	bEnableLuxEvent				: BOOL;
	eEventPriorityBrightness	: E_DALIEventPriority := E_DALIEVENTPRIORITY.Middle;
	nDeadtimeTimerBrightness	: WORD := 1500; // Value in ms, Predefined Value of DALI Standard
	nHysteresisBrightness		: BYTE := 2; // Value in %
	nHysteresisMinBrightness	: BYTE := 10; // Absolute Value, depending on the manufacturer specific resolution
	nReportTimerBrightness		: BYTE := 120; // Value in s, Preset manufacturer value
*)

	//stDaliSetup: SH_Light.ST_DALI_RoomSetup;

END_VAR

VAR CONSTANT
	Sensor_DALI_LINE_NUM: BYTE := 3;
	arrDALI_LINE_NUM_LIGHT: ARRAY[1..2] OF BYTE := [2,1]; //korrekt rækkefølge nødvendig
	arrDALI_LINE_NUM_PENDANTS: ARRAY[1..2] OF BYTE := [0,0]; //korrekt rækkefølge nødvendig. 0 = ingen pendler
END_VAR
VAR PERSISTENT
	stPirSensorData: SH_Light.ST_DALI_Sensor;
	arrstTuneDataGruppe: ARRAY [1..2] OF SH_Light.ST_TuneData_EX;
END_VAR

A_Buttons();
A_LightCtrl();
A_Sensor();

ACTION A_Buttons:
bTopButtonZone1		:= GVL_EnOcean.strEnOceanSwitch_Gang_4_330.bT2_OFF OR bTopButtonZone1_Visu;
bBottomButtonZone1	:= GVL_EnOcean.strEnOceanSwitch_Gang_4_330.bT2_ON OR bBottomButtonZone1_Visu;
END_ACTION

ACTION A_LightCtrl:
bNeighborRoomsPir	:= P_Gang_4_308.stPirSensorData.bPrc      OR
						P_Rum_4_324.stPirSensorData.bPrc      OR
						P_Rum_4_325.stPirSensorData.bPrc      OR
						P_Rum_4_329.stPirSensorData.bPrc;


//gruppe 3
arrfbLysGruppe[1]( 
	nZoneID:= 1, 
	bButtonZone1:= bTopButtonZone1,
	bBottomButtonZone1 := bBottomButtonZone1, 
	bButtonZone2:= bButtonZone2,
	bNeighborRoomsPir	:=	bNeighborRoomsPir,
	fLuxOn:= fLuxOn, 
	fLuxDim:= fLuxDim, 
	tPIRDim:= tPIRDim, 
	tPIROff:= tPIROff, 
	fOffsetSec:= fOffsetSec, 
	bReInit:= , 
	stDaliSetup:= arrstDaliSetupGruppe[1], 
	ipCommunication_Prim:= P_DALI_Background.arrfbKL6821Communication[arrDALI_LINE_NUM_LIGHT[1]], 
	ipCommunication_Sec:= P_DALI_Background.arrfbKL6821Communication[arrDALI_LINE_NUM_LIGHT[1]], //samme som lyslinjen, hvis den ikke eksisterer
	ipCommunication_Supl:= P_DALI_Background.arrfbKL6821Communication[arrDALI_LINE_NUM_LIGHT[1]],//samme som lyslinjen, hvis den ikke eksisterer 
	fMinOutputPowerLevelRoom:= 15, 
	fMaxOutputPowerLevelRoom:= 100, 
	nCycleTimeInMS:= 10 , 
	bRunTuning:= arrRunTuningGruppe[1], 
	bOccupiedRoom=> , 
	bError_Prim=> , 
	nError_Prim=> , 
	stTuneData:=arrstTuneDataGruppe[1] , 
	stPirSensorData:= stPirSensorData, 					//samme sensordata
	stLiveData:= arrstLiveDataGruppe[1]);

//gruppe 13
arrfbLysGruppe[2]( 
	nZoneID:= 1, 
	bButtonZone1:= bTopButtonZone1,
	bBottomButtonZone1 := bBottomButtonZone1, 
	bButtonZone2:= bButtonZone2,
	bNeighborRoomsPir	:=	bNeighborRoomsPir,
	fLuxOn:= fLuxOn, 
	fLuxDim:= fLuxDim, 
	tPIRDim:= tPIRDim, 
	tPIROff:= tPIROff, 
	fOffsetSec:= fOffsetSec, 
	bReInit:= , 
	stDaliSetup:= arrstDaliSetupGruppe[2], 
	ipCommunication_Prim:= P_DALI_Background.arrfbKL6821Communication[arrDALI_LINE_NUM_LIGHT[2]], 
	ipCommunication_Sec:= P_DALI_Background.arrfbKL6821Communication[arrDALI_LINE_NUM_LIGHT[2]], //samme som lyslinjen, hvis den ikke eksisterer
	ipCommunication_Supl:= P_DALI_Background.arrfbKL6821Communication[arrDALI_LINE_NUM_LIGHT[2]], //samme som lyslinjen, hvis den ikke eksisterer 
	fMinOutputPowerLevelRoom:= 15, 
	fMaxOutputPowerLevelRoom:= 100, 
	nCycleTimeInMS:= 10 , 
	bRunTuning:= arrRunTuningGruppe[2], 
	bOccupiedRoom=> , 
	bError_Prim=> , 
	nError_Prim=> , 
	stTuneData:=arrstTuneDataGruppe[2] , 
	stPirSensorData:= stPirSensorData, 					//samme sensordata
	stLiveData:= arrstLiveDataGruppe[2]);
END_ACTION

ACTION A_Sensor:

fbSensor.ipCommunication := P_DALI_Background.arrfbKL6821Communication[Sensor_DALI_LINE_NUM];

//only 1 sensor
fbSensor(
	byShrtAdr:= bySensorAddr,
	bInitialize:= bInitialize, 
	DALI_LINE_NUM:= Sensor_DALI_LINE_NUM, 
 	//bCancelHoldTimerOccupancy:= bCancelHoldTimerOccupancy, 
	stSensorSetup := stDaliSensorSetup,
	bInitErr=> bInitErr, 
	bInitDone=> bInitDone,
	stPirSensorData:= stPirSensorData, 
	arrSensorScales:= arrSensorScales);


(*//several sensors	
fbSensor(
	arrShrtAdr:= arrSensorAddr,
	bInitialize:= bInitialize, 
	DALI_LINE_NUM:= Sensor_DALI_LINE_NUM, 
 	//bCancelHoldTimerOccupancy:= bCancelHoldTimerOccupancy, 
	stSensorSetup := stDaliSensorSetup,
	arrInitErr=> arrInitErr, 
	arrInitDone=> arrInitDone,
	stPirSensorData:= stPirSensorData, 
	arrSensorScales:= arrSensorScales);
	*)
END_ACTION

END_PROGRAM

// ---- POUs/Alle_Rum/Gange/Gang_4_308_2linjerLampe/P_Gang_4_308.TcPOU
PROGRAM P_Gang_4_308
VAR
(*Gangen består af to lysgrupper - 5 og 14 - på to forskellige DALI-linjer - 2 og 1 henh..
Begge grupper afhænger af samme PIR-input - pir-adr. 6, 7, 8, 9 og 10 - på DALI-linje 2.
Derfor oprettes to adskilte reguleringer med samme PV. Dvs., at knapfunktion og pirfunktion forbliver den samme.

En anden del af af hele gangen styres fra AH4_3. De to dele nabostyres med PIR-signaler over modbus-kommunikation*)

	arrfbLysGruppe			: ARRAY [1..2] OF FB_Light_Type_B;
	arrstDaliSetupGruppe	: ARRAY[1..2] OF SH_Light.ST_DALI_RoomSetup := 
	
													[(	byShrtAdr_Prim := 29, 
														byGrpAdr_Prim := 5, 
														eMod_Prim := E_DALIAddressType.Group, 
														byShrtAdr_Sec := 1, 
														byGrpAdr_Sec := 1, 
														eMod_Sec := E_DALIAddressType.Short, 
														byShrtAdr_Supl := 1, 
														DALI_LINE_NUM_PRIM := arrDALI_LINE_NUM_LIGHT[1], 
														DALI_LINE_NUM_SEC := 0, //0 = ingen zonestyring/vinduerække
														DALI_LINE_NUM_SUPL := arrDALI_LINE_NUM_PENDANTS[1]),
														
													(	byShrtAdr_Prim := 51, 
														byGrpAdr_Prim := 14, 
														eMod_Prim := E_DALIAddressType.Group, 
														byShrtAdr_Sec := 1, 
														byGrpAdr_Sec := 1, 
														eMod_Sec := E_DALIAddressType.Short, 
														byShrtAdr_Supl := 1, 
														DALI_LINE_NUM_PRIM := arrDALI_LINE_NUM_LIGHT[2], 
														DALI_LINE_NUM_SEC := 0, 
														DALI_LINE_NUM_SUPL := arrDALI_LINE_NUM_PENDANTS[2])];
														
	arrstLiveDataGruppe		: ARRAY [1..2] OF SH_Light.ST_LiveData;
	//stLiveData AT %MB22	: SH_Light.ST_LiveData;
	
	arrRunTuningGruppe: ARRAY[1..2] OF BOOL;
	
	
	
	bTopButtonZone1			: BOOL;
	bTopButtonZone1_Visu	: BOOL;
	bBottomButtonZone1		: BOOL;
	bBottomButtonZone1_Visu	: BOOL;
	bButtonZone2			: BOOL;
	bNeighborRoomsPir		: BOOL;
	fLuxOn					: REAL := 500;
	fLuxDim					: REAL := 200;
	tPIRDim					: TIME := T#15M;
	tPIROff					: TIME := T#30M;
	fOffsetSec				: REAL := 20;



// Sensor Settings
	//fbSensor					: SH_Light.FB_NIKO_P46xx_1Pcs;
	fbSensor					: SH_Light.FB_NIKO_P46xx_3Pcs;
	//bySensorAddr				: BYTE := 17;
	arrSensorAddr				: ARRAY[1..3] OF BYTE := [7,8,9];
	bInitialize					: BOOL := TRUE;
	stDaliSensorSetup			: ST_DALI_NIKOP46SetupData;
	//bInitErr					: BOOL;
	//bInitDone					: BOOL;
	arrInitErr					: ARRAY [1..3] OF BOOL;
	arrInitDone					: ARRAY [1..3] OF BOOL;
	arrSensorScales				: ARRAY [1..10] OF SH_Light.ST_DALI_SensorScaleMode := [	(fMeassureMaxSensor := 1023, fReadMaxSensor := 1023),
																							(fMeassureMaxSensor := 1023, fReadMaxSensor := 1023),
																							(fMeassureMaxSensor := 1023, fReadMaxSensor := 1023),																						
																						7(())];
	bCancelHoldTimerOccupancy	: BOOL;
(*	eEventPriorityOccupancy		: E_DALIEventPriority := E_DALIEVENTPRIORITY.Middle;
	nHoldTimerOccupancy			: WORD := 5; // Value in s. 	
	nReportTimerOccupancy		: BYTE := 120; // Value in s, Preset manufacturer value
	nDeadtimeTimerOccupancy		: WORD := 100; // Value in ms, Predefined Value of DALI Standard
	bCancelHoldTimerOccupancy	: BOOL;
	nSensitivityOccupancy		: BYTE:= 3; //setting Sensivity (0..4) 0 (Off), 1 (Min), 2(Low), 3(High) and 4 (Max)

	bEnableLuxEvent				: BOOL;
	eEventPriorityBrightness	: E_DALIEventPriority := E_DALIEVENTPRIORITY.Middle;
	nDeadtimeTimerBrightness	: WORD := 1500; // Value in ms, Predefined Value of DALI Standard
	nHysteresisBrightness		: BYTE := 2; // Value in %
	nHysteresisMinBrightness	: BYTE := 10; // Absolute Value, depending on the manufacturer specific resolution
	nReportTimerBrightness		: BYTE := 120; // Value in s, Preset manufacturer value
*)


END_VAR

VAR CONSTANT
	Sensor_DALI_LINE_NUM: BYTE := 3;
	arrDALI_LINE_NUM_LIGHT: ARRAY[1..2] OF BYTE := [2,1]; //korrekt rækkefølge nødvendig
	arrDALI_LINE_NUM_PENDANTS: ARRAY[1..2] OF BYTE := [0,0]; //korrekt rækkefølge nødvendig. 0 = ingen pendler
END_VAR
VAR PERSISTENT
	stPirSensorData: SH_Light.ST_DALI_Sensor;
	arrstTuneDataGruppe: ARRAY [1..2] OF SH_Light.ST_TuneData_EX;
END_VAR

A_Buttons();
A_LightCtrl();
A_Sensor();

ACTION A_Buttons:
bTopButtonZone1		:= bTopButtonZone1_Visu;
bBottomButtonZone1	:= bBottomButtonZone1_Visu;
END_ACTION

ACTION A_LightCtrl:
bNeighborRoomsPir	:=  
						P_Rum_4_324.stPirSensorData.bPrc OR
				     	P_Gang_4_330.stPirSensorData.bPrc OR
						P_Gang_4_334A.stPirSensorData.bPrc OR
                        P_Gang_5_338.stPirSensorData.bPrc;

//gruppe 5
arrfbLysGruppe[1]( 
	nZoneID:= 1, 
	bButtonZone1:= bTopButtonZone1,
	bBottomButtonZone1 := bBottomButtonZone1, 
	bButtonZone2:= bButtonZone2,
	bNeighborRoomsPir	:=	bNeighborRoomsPir,
	fLuxOn:= fLuxOn, 
	fLuxDim:= fLuxDim, 
	tPIRDim:= tPIRDim, 
	tPIROff:= tPIROff, 
	fOffsetSec:= fOffsetSec, 
	bReInit:= , 
	stDaliSetup:= arrstDaliSetupGruppe[1], 
	ipCommunication_Prim:= P_DALI_Background.arrfbKL6821Communication[arrDALI_LINE_NUM_LIGHT[1]], 
	ipCommunication_Sec:= P_DALI_Background.arrfbKL6821Communication[arrDALI_LINE_NUM_LIGHT[1]], //samme som lyslinjen, hvis den ikke eksisterer
	ipCommunication_Supl:= P_DALI_Background.arrfbKL6821Communication[arrDALI_LINE_NUM_LIGHT[1]],//samme som lyslinjen, hvis den ikke eksisterer 
	fMinOutputPowerLevelRoom:= 15, 
	fMaxOutputPowerLevelRoom:= 100, 
	nCycleTimeInMS:= 10 , 
	bRunTuning:= arrRunTuningGruppe[1], 
	bOccupiedRoom=> , 
	bError_Prim=> , 
	nError_Prim=> , 
	stTuneData:=arrstTuneDataGruppe[1] , 
	stPirSensorData:= stPirSensorData, 					//samme sensordata
	stLiveData:= arrstLiveDataGruppe[1]);

//gruppe 14	
arrfbLysGruppe[2]( 
	nZoneID:= 1, 
	bButtonZone1:= bTopButtonZone1,
	bBottomButtonZone1 := bBottomButtonZone1, 
	bButtonZone2:= bButtonZone2,
	bNeighborRoomsPir	:=	bNeighborRoomsPir,
	fLuxOn:= fLuxOn, 
	fLuxDim:= fLuxDim, 
	tPIRDim:= tPIRDim, 
	tPIROff:= tPIROff, 
	fOffsetSec:= fOffsetSec, 
	bReInit:= , 
	stDaliSetup:= arrstDaliSetupGruppe[2], 
	ipCommunication_Prim:= P_DALI_Background.arrfbKL6821Communication[arrDALI_LINE_NUM_LIGHT[2]], 
	ipCommunication_Sec:= P_DALI_Background.arrfbKL6821Communication[arrDALI_LINE_NUM_LIGHT[2]], //samme som lyslinjen, hvis den ikke eksisterer
	ipCommunication_Supl:= P_DALI_Background.arrfbKL6821Communication[arrDALI_LINE_NUM_LIGHT[2]], //samme som lyslinjen, hvis den ikke eksisterer 
	fMinOutputPowerLevelRoom:= 15, 
	fMaxOutputPowerLevelRoom:= 100, 
	nCycleTimeInMS:= 10 , 
	bRunTuning:= arrRunTuningGruppe[2], 
	bOccupiedRoom=> , 
	bError_Prim=> , 
	nError_Prim=> , 
	stTuneData:=arrstTuneDataGruppe[2] , 
	stPirSensorData:= stPirSensorData, 					//samme sensordata
	stLiveData:= arrstLiveDataGruppe[2]);
END_ACTION

ACTION A_Sensor:

fbSensor.ipCommunication := P_DALI_Background.arrfbKL6821Communication[Sensor_DALI_LINE_NUM];

(*//only 1 sensor
fbSensor(
	byShrtAdr:= bySensorAddr,
	bInitialize:= bInitialize, 
	DALI_LINE_NUM:= Sensor_DALI_LINE_NUM, 
 	//bCancelHoldTimerOccupancy:= bCancelHoldTimerOccupancy, 
	stSensorSetup := stDaliSensorSetup,
	bInitErr=> bInitErr, 
	bInitDone=> bInitDone,
	stPirSensorData:= stPirSensorData, 
	arrSensorScales:= arrSensorScales);
	*)

//several sensors	
fbSensor(
	arrShrtAdr:= arrSensorAddr,
	bInitialize:= bInitialize, 
	DALI_LINE_NUM:= Sensor_DALI_LINE_NUM, 
 	//bCancelHoldTimerOccupancy:= bCancelHoldTimerOccupancy, 
	stSensorSetup := stDaliSensorSetup,
	arrInitErr=> arrInitErr, 
	arrInitDone=> arrInitDone,
	stPirSensorData:= stPirSensorData, 
	arrSensorScales:= arrSensorScales);
END_ACTION

END_PROGRAM

// ---- POUs/Alle_Rum/Gange/Gang_4_310A/P_Gang_4_310A.TcPOU
PROGRAM P_Gang_4_310A
VAR
//Light

(*Toiletgangen er oprettet som type B i tilfælde af, at gangen skal nabostyres af toiletter mv. i fremtiden.
For nu er der ingen pirsignaler fra toiletter til PLC*)

	fbLys		: FB_Light_Type_B;
	
	stDaliSetup	: SH_Light.ST_DALI_RoomSetup := (		byShrtAdr_Prim := 34, 
														byGrpAdr_Prim := 5, 
														eMod_Prim := E_DALIAddressType.Group, 
														byShrtAdr_Sec := 1, 
														byGrpAdr_Sec := 1, 
														eMod_Sec := E_DALIAddressType.Short, 
														byShrtAdr_Supl := 1, 
														DALI_LINE_NUM_PRIM := DALI_LINE_NUM_LIGHT, 
														DALI_LINE_NUM_SEC := 0, 
														DALI_LINE_NUM_SUPL := DALI_LINE_NUM_PENDANTS);
	stLiveData				: SH_Light.ST_LiveData;
	//stLiveData AT %MB22	: SH_Light.ST_LiveData;
	bTopButtonZone1			: BOOL;
	bTopButtonZone1_Visu		: BOOL;
	bBottomButtonZone1		: BOOL;
	bBottomButtonZone1_Visu	: BOOL;
	bButtonZone2			: BOOL;
	bNeighborRoomsPir		: BOOL;
	fLuxOn					: REAL := 500;
	fLuxDim					: REAL := 200;
	tPIRDim					: TIME := T#15M;
	tPIROff					: TIME := T#30M;
	fOffsetSec				: REAL := 20;

	bRunTuning: BOOL;

// Sensor Settings
	fbSensor					: SH_Light.FB_NIKO_P46xx_1Pcs;	
	//fbSensor					: SH_Light.FB_NIKO_P46xx_2Pcs;
	bySensorAddr				: BYTE := 1;
	//arrSensorAddr				: ARRAY[1..2] OF BYTE := [12,13];
	bInitialize					: BOOL := TRUE;
	stDaliSensorSetup			: ST_DALI_NIKOP46SetupData;
	bInitErr					: BOOL;
	bInitDone					: BOOL;
	//arrInitErr					: ARRAY [1..2] OF BOOL;
	//arrInitDone					: ARRAY [1..2] OF BOOL;
	arrSensorScales				: ARRAY [1..10] OF SH_Light.ST_DALI_SensorScaleMode := [	(fMeassureMaxSensor := 1023, fReadMaxSensor := 1023),
																						9(())];
	bCancelHoldTimerOccupancy	: BOOL;
(*	eEventPriorityOccupancy		: E_DALIEventPriority := E_DALIEVENTPRIORITY.Middle;
	nHoldTimerOccupancy			: WORD := 5; // Value in s. 	
	nReportTimerOccupancy		: BYTE := 120; // Value in s, Preset manufacturer value
	nDeadtimeTimerOccupancy		: WORD := 100; // Value in ms, Predefined Value of DALI Standard
	bCancelHoldTimerOccupancy	: BOOL;
	nSensitivityOccupancy		: BYTE:= 3; //setting Sensivity (0..4) 0 (Off), 1 (Min), 2(Low), 3(High) and 4 (Max)

	bEnableLuxEvent				: BOOL;
	eEventPriorityBrightness	: E_DALIEventPriority := E_DALIEVENTPRIORITY.Middle;
	nDeadtimeTimerBrightness	: WORD := 1500; // Value in ms, Predefined Value of DALI Standard
	nHysteresisBrightness		: BYTE := 2; // Value in %
	nHysteresisMinBrightness	: BYTE := 10; // Absolute Value, depending on the manufacturer specific resolution
	nReportTimerBrightness		: BYTE := 120; // Value in s, Preset manufacturer value
*)

END_VAR

VAR CONSTANT
	Sensor_DALI_LINE_NUM	: BYTE := 3;
	DALI_LINE_NUM_LIGHT		: BYTE := 3;
	DALI_LINE_NUM_PENDANTS	: BYTE := 0;
END_VAR
VAR PERSISTENT
	stPirSensorData: SH_Light.ST_DALI_Sensor;
	stTuneData: SH_Light.ST_TuneData_EX;
END_VAR

A_Buttons();
A_LightCtrl();
A_Sensor();

ACTION A_Buttons:
bTopButtonZone1		:=  bTopButtonZone1_Visu;
bBottomButtonZone1	:=  bBottomButtonZone1_Visu;
END_ACTION

ACTION A_LightCtrl:
bNeighborRoomsPir	:= 0; //evt. nabostyring
						
fbLys(
	nZoneID:= 1, 
	bButtonZone1:= bTopButtonZone1,
	bBottomButtonZone1 := bBottomButtonZone1, 
	bButtonZone2:= bButtonZone2,
	bNeighborRoomsPir	:=	bNeighborRoomsPir,
	fLuxOn:= fLuxOn, 
	fLuxDim:= fLuxDim, 
	tPIRDim:= tPIRDim, 
	tPIROff:= tPIROff, 
	fOffsetSec:= fOffsetSec, 
	bReInit:= , 
	stDaliSetup:= stDaliSetup, 
	ipCommunication_Prim:= P_DALI_Background.arrfbKL6821Communication[DALI_LINE_NUM_LIGHT], 
	ipCommunication_Sec:= P_DALI_Background.arrfbKL6821Communication[DALI_LINE_NUM_LIGHT], 
	ipCommunication_Supl:= P_DALI_Background.arrfbKL6821Communication[DALI_LINE_NUM_LIGHT], 
	fMinOutputPowerLevelRoom:= 15, 
	fMaxOutputPowerLevelRoom:= 100, 
	nCycleTimeInMS:= 10 , 
	bRunTuning:= bRunTuning, 
	bOccupiedRoom=> , 
	bError_Prim=> , 
	nError_Prim=> , 
	stTuneData:=stTuneData , 
	stPirSensorData:= stPirSensorData, 
	stLiveData:= stLiveData);
END_ACTION

ACTION A_Sensor:

fbSensor.ipCommunication := P_DALI_Background.arrfbKL6821Communication[Sensor_DALI_LINE_NUM];

//Only 1 sensor
fbSensor(
	byShrtAdr:= bySensorAddr,
	bInitialize:= bInitialize, 
	DALI_LINE_NUM:= Sensor_DALI_LINE_NUM, 
 	//bCancelHoldTimerOccupancy:= bCancelHoldTimerOccupancy, 
	stSensorSetup := stDaliSensorSetup,
	bInitErr=> bInitErr, 
	bInitDone=> bInitDone,
	stPirSensorData:= stPirSensorData, 
	arrSensorScales:= arrSensorScales);

(*//Several sensors
fbSensor(
	arrShrtAdr:= arrSensorAddr,
	bInitialize:= bInitialize, 
	DALI_LINE_NUM:= Sensor_DALI_LINE_NUM, 
 	//bCancelHoldTimerOccupancy:= bCancelHoldTimerOccupancy, 
	stSensorSetup := stDaliSensorSetup,
	arrInitErr=> arrInitErr, 
	arrInitDone=> arrInitDone,
	stPirSensorData:= stPirSensorData, 
	arrSensorScales:= arrSensorScales);
	*)
END_ACTION

END_PROGRAM

// ---- POUs/Alle_Rum/Rum_Med_DALI_Pir/P_Lys_Grp0.TcPOU
PROGRAM P_Lys_Grp0
VAR
	fbLight_GRP0: FB_DALILgtActr_EX;
	eMod: SH_Light.E_DALIAddressType := SH_Light.E_DALIAddressType.Group;
	fSttupCtrlVal: REAL;
	fMinCtrlVal: REAL := 0;
	fMaxCtrlVal: REAL := 100;
	fLgtOffset: REAL := 5;
	eFadeTime: SH_Light.E_DALIFadeTime := SH_Light.E_DALIFadeTime.T02000ms;
	eFadeRate: SH_Light.E_DALIFadeRate := SH_Light.E_DALIFadeRate.N063StepsPerSec;
	uiBlinkTi: UINT := 2;
	uiOffDly: UINT := 0;
	uiPollActLgtLvl: UINT := 30;
	bReInit: BOOL;
	nCycleTimeInMS: UDINT := 10;
	stLgtCmd: SH_Light.ST_LgtCmd;
END_VAR

VAR CONSTANT
	DALI_LINE_NUM: BYTE := 1;
END_VAR

fbLight_GRP0.ipDALICommunication := P_DALI_Background.arrfbKL6821Communication[DALI_LINE_NUM];
fbLight_GRP0(
    byShrtAdr := 6,
    byGrpAdr := 1,
    eMod := eMod,
    fSttupCtrlVal := fSttupCtrlVal,
    fMinCtrlVal := fMinCtrlVal,
    fMaxCtrlVal := fMaxCtrlVal,
    fLgtOffset := fLgtOffset,
    eFadeTime := eFadeTime,
    eFadeRate := eFadeRate,
    uiBlinkTi := uiBlinkTi,
    uiOffDly := uiOffDly,
    uiPollActLgtLvl := uiPollActLgtLvl,
    bReInit := bReInit,
    nCycleTimeInMS := nCycleTimeInMS,
    stLgtCmd := stLgtCmd,
    DALI_LINE_NUM := DALI_LINE_NUM); // FB_DALILgtActr_EX

END_PROGRAM

// ---- POUs/Alle_Rum/Rum_Med_DALI_Pir/Rum_5_341/P_Rum_5_341.TcPOU
PROGRAM P_Rum_5_341
VAR
//Light

	fbLys		: FB_Light_Type_A;
	
	stDaliSetup	: SH_Light.ST_DALI_RoomSetup := (		byShrtAdr_Prim := 5, 
														byGrpAdr_Prim := 2, 
														eMod_Prim := E_DALIAddressType.Group, 
														byShrtAdr_Sec := 1, 
														byGrpAdr_Sec := 1, 
														eMod_Sec := E_DALIAddressType.Short, 
														byShrtAdr_Supl := 1, 
														DALI_LINE_NUM_PRIM := DALI_LINE_NUM_LIGHT, 
														DALI_LINE_NUM_SEC := 0, //0 = ingen zonestyring/vinduerække
														DALI_LINE_NUM_SUPL := DALI_LINE_NUM_PENDANTS);
	stLiveData				: SH_Light.ST_LiveData;
	//stLiveData AT %MB22	: SH_Light.ST_LiveData;
	bTopButtonZone1			: BOOL;
	bTopButtonZone1_Visu	: BOOL;
	bBottomButtonZone1		: BOOL;
	bBottomButtonZone1_Visu	: BOOL;
	bButtonZone2			: BOOL;
	fLuxOn					: REAL := 500;
	fLuxDim					: REAL := 200;
	tPIRDim					: TIME := T#15M;
	tPIROff					: TIME := T#30M;
	fOffsetSec				: REAL := 20;
	bOccupiedRoom			: BOOL;

	bRunTuning				: BOOL;
	
// Sensor Settings
	fbSensor					: SH_Light.FB_NIKO_P46xx_1Pcs;
	//fbSensor					: SH_Light.FB_NIKO_P46xx_2Pcs;
	bySensorAddr				: BYTE := 2;
	//arrSensorAddr				: ARRAY[1..2] OF BYTE := [9,10];
	bInitialize					: BOOL := TRUE;
	stDaliSensorSetup			: ST_DALI_NIKOP46SetupData;
	bInitErr					: BOOL;
	bInitDone					: BOOL;
	//arrInitErr					: ARRAY [1..2] OF BOOL;
	//arrInitDone					: ARRAY [1..2] OF BOOL;
	arrSensorScales				: ARRAY [1..10] OF SH_Light.ST_DALI_SensorScaleMode := [	(fMeassureMaxSensor := 1023, fReadMaxSensor := 1023),
																						9(())];
	bCancelHoldTimerOccupancy	: BOOL;
(*	eEventPriorityOccupancy		: E_DALIEventPriority := E_DALIEVENTPRIORITY.Middle;
	nHoldTimerOccupancy			: WORD := 5; // Value in s. 	
	nReportTimerOccupancy		: BYTE := 120; // Value in s, Preset manufacturer value
	nDeadtimeTimerOccupancy		: WORD := 100; // Value in ms, Predefined Value of DALI Standard
	bCancelHoldTimerOccupancy	: BOOL;
	nSensitivityOccupancy		: BYTE:= 3; //setting Sensivity (0..4) 0 (Off), 1 (Min), 2(Low), 3(High) and 4 (Max)

	bEnableLuxEvent				: BOOL;
	eEventPriorityBrightness	: E_DALIEventPriority := E_DALIEVENTPRIORITY.Middle;
	nDeadtimeTimerBrightness	: WORD := 1500; // Value in ms, Predefined Value of DALI Standard
	nHysteresisBrightness		: BYTE := 2; // Value in %
	nHysteresisMinBrightness	: BYTE := 10; // Absolute Value, depending on the manufacturer specific resolution
	nReportTimerBrightness		: BYTE := 120; // Value in s, Preset manufacturer value
*)

END_VAR

VAR CONSTANT
	Sensor_DALI_LINE_NUM	: BYTE := 2;
	DALI_LINE_NUM_LIGHT		: BYTE := 1;
	DALI_LINE_NUM_PENDANTS	: BYTE := 0; //0=ingen pendler
END_VAR
VAR PERSISTENT
	stPirSensorData: SH_Light.ST_DALI_Sensor;
	stTuneData: SH_Light.ST_TuneData_EX;
END_VAR

A_Buttons();
A_LightCtrl();
A_Sensor();

ACTION A_Buttons:
bTopButtonZone1		:= GVL_EnOcean.strEnOceanSwitch_Rum_5_341.bT1_ON OR bTopButtonZone1_Visu;
bBottomButtonZone1	:= GVL_EnOcean.strEnOceanSwitch_Rum_5_341.bT1_OFF OR bBottomButtonZone1_Visu;
END_ACTION

ACTION A_LightCtrl:

fbLys(
	nZoneID:= 1, 
	bButtonZone1:= bTopButtonZone1,
	bBottomButtonZone1 := bBottomButtonZone1, 
	bButtonZone2:= bButtonZone2, 
	fLuxOn:= fLuxOn, 
	fLuxDim:= fLuxDim, 
	tPIRDim:= tPIRDim, 
	tPIROff:= tPIROff, 
	fOffsetSec:= fOffsetSec, 
	bReInit:= , 
	stDaliSetup:= stDaliSetup, 
	ipCommunication_Prim:= P_DALI_Background.arrfbKL6821Communication[DALI_LINE_NUM_LIGHT], 
	ipCommunication_Sec:= P_DALI_Background.arrfbKL6821Communication[DALI_LINE_NUM_LIGHT], 
	ipCommunication_Supl:= P_DALI_Background.arrfbKL6821Communication[DALI_LINE_NUM_LIGHT], 
	fMinOutputPowerLevelRoom:= 15, 
	fMaxOutputPowerLevelRoom:= 100, 
	nCycleTimeInMS:= 10 , 
	bRunTuning:= bRunTuning, 
	bOccupiedRoom=> bOccupiedRoom, 
	bError_Prim=> , 
	nError_Prim=> , 
	stTuneData:=stTuneData , 
	stPirSensorData:= stPirSensorData, 
	stLiveData:= stLiveData);
END_ACTION

ACTION A_Sensor:

fbSensor.ipCommunication := P_DALI_Background.arrfbKL6821Communication[Sensor_DALI_LINE_NUM];


fbSensor(
	byShrtAdr:= bySensorAddr,
	bInitialize:= bInitialize, 
	DALI_LINE_NUM:= Sensor_DALI_LINE_NUM, 
 	//bCancelHoldTimerOccupancy:= bCancelHoldTimerOccupancy, 
	stSensorSetup := stDaliSensorSetup,
	bInitErr=> bInitErr, 
	bInitDone=> bInitDone,
	stPirSensorData:= stPirSensorData, 
	arrSensorScales:= arrSensorScales);

(*
fbSensor(
	arrShrtAdr:= arrSensorAddr,
	bInitialize:= bInitialize, 
	DALI_LINE_NUM:= Sensor_DALI_LINE_NUM, 
 	//bCancelHoldTimerOccupancy:= bCancelHoldTimerOccupancy, 
	stSensorSetup := stDaliSensorSetup,
	arrInitErr=> arrInitErr, 
	arrInitDone=> arrInitDone,
	stPirSensorData:= stPirSensorData, 
	arrSensorScales:= arrSensorScales);
	*)
END_ACTION

END_PROGRAM

// ---- POUs/Alle_Rum/Rum_Med_DALI_Pir/Rum_5_343_2linjerPIR/P_Rum_5_343.TcPOU
PROGRAM P_Rum_5_343
VAR
//Light

	fbLys		: FB_Light_Type_A;
	
	stDaliSetup	: SH_Light.ST_DALI_RoomSetup := (		byShrtAdr_Prim := 7, 
														byGrpAdr_Prim := 3, 
														eMod_Prim := E_DALIAddressType.Group, 
														byShrtAdr_Sec := 1, 
														byGrpAdr_Sec := 1, 
														eMod_Sec := E_DALIAddressType.Short, 
														byShrtAdr_Supl := 1, 
														DALI_LINE_NUM_PRIM := DALI_LINE_NUM_LIGHT, 
														DALI_LINE_NUM_SEC := 0, //0 = ingen zonestyring/vinduerække
														DALI_LINE_NUM_SUPL := DALI_LINE_NUM_PENDANTS);
	stLiveData				: SH_Light.ST_LiveData;
	//stLiveData AT %MB22	: SH_Light.ST_LiveData;
	bTopButtonZone1			: BOOL;
	bTopButtonZone1_Visu	: BOOL;
	bBottomButtonZone1		: BOOL;
	bBottomButtonZone1_Visu	: BOOL;
	bButtonZone2			: BOOL;
	fLuxOn					: REAL := 500;
	fLuxDim					: REAL := 200;
	tPIRDim					: TIME := T#15M;
	tPIROff					: TIME := T#30M;
	fOffsetSec				: REAL := 20;
	bOccupiedRoom			: BOOL;

	bRunTuning				: BOOL;
	
// Sensor Settings
	fbSensor					: SH_Light.FB_NIKO_P46xx_1Pcs;
	//fbSensor					: SH_Light.FB_NIKO_P46xx_2Pcs;
	bySensorAddr				: BYTE := 3;
	//arrSensorAddr				: ARRAY[1..2] OF BYTE := [9,10];
	bInitialize					: BOOL := TRUE;
	stDaliSensorSetup			: ST_DALI_NIKOP46SetupData;
	bInitErr					: BOOL;
	bInitDone					: BOOL;
	//arrInitErr					: ARRAY [1..2] OF BOOL;
	//arrInitDone					: ARRAY [1..2] OF BOOL;
	arrSensorScales				: ARRAY [1..10] OF SH_Light.ST_DALI_SensorScaleMode := [	(fMeassureMaxSensor := 1023, fReadMaxSensor := 1023),
																						9(())];
	bCancelHoldTimerOccupancy	: BOOL;
(*	eEventPriorityOccupancy		: E_DALIEventPriority := E_DALIEVENTPRIORITY.Middle;
	nHoldTimerOccupancy			: WORD := 5; // Value in s. 	
	nReportTimerOccupancy		: BYTE := 120; // Value in s, Preset manufacturer value
	nDeadtimeTimerOccupancy		: WORD := 100; // Value in ms, Predefined Value of DALI Standard
	bCancelHoldTimerOccupancy	: BOOL;
	nSensitivityOccupancy		: BYTE:= 3; //setting Sensivity (0..4) 0 (Off), 1 (Min), 2(Low), 3(High) and 4 (Max)

	bEnableLuxEvent				: BOOL;
	eEventPriorityBrightness	: E_DALIEventPriority := E_DALIEVENTPRIORITY.Middle;
	nDeadtimeTimerBrightness	: WORD := 1500; // Value in ms, Predefined Value of DALI Standard
	nHysteresisBrightness		: BYTE := 2; // Value in %
	nHysteresisMinBrightness	: BYTE := 10; // Absolute Value, depending on the manufacturer specific resolution
	nReportTimerBrightness		: BYTE := 120; // Value in s, Preset manufacturer value
*)

END_VAR

VAR CONSTANT
	Sensor_DALI_LINE_NUM	: BYTE := 2;
	DALI_LINE_NUM_LIGHT		: BYTE := 1;
	DALI_LINE_NUM_PENDANTS	: BYTE := 0; //0=ingen pendler
END_VAR
VAR PERSISTENT
	stPirSensorData: SH_Light.ST_DALI_Sensor;
	stTuneData: SH_Light.ST_TuneData_EX;
END_VAR

A_Buttons();
A_LightCtrl();
A_Sensor();

ACTION A_Buttons:
bTopButtonZone1		:= GVL_EnOcean.strEnOceanSwitch_Rum_5_343.bT1_ON OR bTopButtonZone1_Visu;
bBottomButtonZone1	:= GVL_EnOcean.strEnOceanSwitch_Rum_5_343.bT1_OFF OR bBottomButtonZone1_Visu;
END_ACTION

ACTION A_LightCtrl:

fbLys(
	nZoneID:= 1, 
	bButtonZone1:= bTopButtonZone1,
	bBottomButtonZone1 := bBottomButtonZone1, 
	bButtonZone2:= bButtonZone2, 
	fLuxOn:= fLuxOn, 
	fLuxDim:= fLuxDim, 
	tPIRDim:= tPIRDim, 
	tPIROff:= tPIROff, 
	fOffsetSec:= fOffsetSec, 
	bReInit:= , 
	stDaliSetup:= stDaliSetup, 
	ipCommunication_Prim:= P_DALI_Background.arrfbKL6821Communication[DALI_LINE_NUM_LIGHT], 
	ipCommunication_Sec:= P_DALI_Background.arrfbKL6821Communication[DALI_LINE_NUM_LIGHT], 
	ipCommunication_Supl:= P_DALI_Background.arrfbKL6821Communication[DALI_LINE_NUM_LIGHT], 
	fMinOutputPowerLevelRoom:= 15, 
	fMaxOutputPowerLevelRoom:= 100, 
	nCycleTimeInMS:= 10 , 
	bRunTuning:= bRunTuning, 
	bOccupiedRoom=> bOccupiedRoom, 
	bError_Prim=> , 
	nError_Prim=> , 
	stTuneData:=stTuneData , 
	stPirSensorData:= stPirSensorData, 
	stLiveData:= stLiveData);
END_ACTION

ACTION A_Sensor:

fbSensor.ipCommunication := P_DALI_Background.arrfbKL6821Communication[Sensor_DALI_LINE_NUM];


fbSensor(
	byShrtAdr:= bySensorAddr,
	bInitialize:= bInitialize, 
	DALI_LINE_NUM:= Sensor_DALI_LINE_NUM, 
 	//bCancelHoldTimerOccupancy:= bCancelHoldTimerOccupancy, 
	stSensorSetup := stDaliSensorSetup,
	bInitErr=> bInitErr, 
	bInitDone=> bInitDone,
	stPirSensorData:= stPirSensorData, 
	arrSensorScales:= arrSensorScales);

(*
fbSensor(
	arrShrtAdr:= arrSensorAddr,
	bInitialize:= bInitialize, 
	DALI_LINE_NUM:= Sensor_DALI_LINE_NUM, 
 	//bCancelHoldTimerOccupancy:= bCancelHoldTimerOccupancy, 
	stSensorSetup := stDaliSensorSetup,
	arrInitErr=> arrInitErr, 
	arrInitDone=> arrInitDone,
	stPirSensorData:= stPirSensorData, 
	arrSensorScales:= arrSensorScales);
	*)
END_ACTION

END_PROGRAM

// ---- POUs/Alle_Rum/Rum_Med_DALI_Pir/Rum_5_350B_short/P_Rum_5_350B.TcPOU
PROGRAM P_Rum_5_350B
VAR
//Light

	fbLys		: FB_Light_Type_A;
	
	stDaliSetup	: SH_Light.ST_DALI_RoomSetup := (		byShrtAdr_Prim := 18, 
														byGrpAdr_Prim := 0, 
														eMod_Prim := E_DALIAddressType.Short, 
														byShrtAdr_Sec := 0, 
														byGrpAdr_Sec := 0, 
														eMod_Sec := E_DALIAddressType.group, 
														byShrtAdr_Supl := 1, 
														DALI_LINE_NUM_PRIM := DALI_LINE_NUM_LIGHT, 
														DALI_LINE_NUM_SEC := 0, //0 = ingen zonestyring/vinduerække
														DALI_LINE_NUM_SUPL := DALI_LINE_NUM_PENDANTS);
	stLiveData				: SH_Light.ST_LiveData;
	//stLiveData AT %MB22	: SH_Light.ST_LiveData;
	bTopButtonZone1			: BOOL;
	bTopButtonZone1_Visu	: BOOL;
	bBottomButtonZone1		: BOOL;
	bBottomButtonZone1_Visu	: BOOL;
	bButtonZone2			: BOOL;
	fLuxOn					: REAL := 500;
	fLuxDim					: REAL := 200;
	tPIRDim					: TIME := T#15M;
	tPIROff					: TIME := T#30M;
	fOffsetSec				: REAL := 20;
	bOccupiedRoom			: BOOL;

	bRunTuning				: BOOL;
	
// Sensor Settings
	fbSensor					: SH_Light.FB_NIKO_P46xx_1Pcs;
	//fbSensor					: SH_Light.FB_NIKO_P46xx_2Pcs;
	bySensorAddr				: BYTE := 2;
	//arrSensorAddr				: ARRAY[1..2] OF BYTE := [9,10];
	bInitialize					: BOOL := TRUE;
	stDaliSensorSetup			: ST_DALI_NIKOP46SetupData;
	bInitErr					: BOOL;
	bInitDone					: BOOL;
	//arrInitErr					: ARRAY [1..2] OF BOOL;
	//arrInitDone					: ARRAY [1..2] OF BOOL;
	arrSensorScales				: ARRAY [1..10] OF SH_Light.ST_DALI_SensorScaleMode := [	(fMeassureMaxSensor := 1023, fReadMaxSensor := 1023),
																						9(())];
	bCancelHoldTimerOccupancy	: BOOL;
(*	eEventPriorityOccupancy		: E_DALIEventPriority := E_DALIEVENTPRIORITY.Middle;
	nHoldTimerOccupancy			: WORD := 5; // Value in s. 	
	nReportTimerOccupancy		: BYTE := 120; // Value in s, Preset manufacturer value
	nDeadtimeTimerOccupancy		: WORD := 100; // Value in ms, Predefined Value of DALI Standard
	bCancelHoldTimerOccupancy	: BOOL;
	nSensitivityOccupancy		: BYTE:= 3; //setting Sensivity (0..4) 0 (Off), 1 (Min), 2(Low), 3(High) and 4 (Max)

	bEnableLuxEvent				: BOOL;
	eEventPriorityBrightness	: E_DALIEventPriority := E_DALIEVENTPRIORITY.Middle;
	nDeadtimeTimerBrightness	: WORD := 1500; // Value in ms, Predefined Value of DALI Standard
	nHysteresisBrightness		: BYTE := 2; // Value in %
	nHysteresisMinBrightness	: BYTE := 10; // Absolute Value, depending on the manufacturer specific resolution
	nReportTimerBrightness		: BYTE := 120; // Value in s, Preset manufacturer value
*)

END_VAR

VAR CONSTANT
	Sensor_DALI_LINE_NUM	: BYTE := 1;
	DALI_LINE_NUM_LIGHT		: BYTE := 1;
	DALI_LINE_NUM_PENDANTS	: BYTE := 0; //0=ingen pendler
END_VAR
VAR PERSISTENT
	stPirSensorData: SH_Light.ST_DALI_Sensor;
	stTuneData: SH_Light.ST_TuneData_EX;
END_VAR

A_Buttons();
A_LightCtrl();
A_Sensor();

ACTION A_Buttons:
//bTopButtonZone1		:= GVL_EnOcean.strEnOceanSwitch_Rum_5_350B.bT2_ON OR bTopButtonZone1_Visu;
//bBottomButtonZone1	:= GVL_EnOcean.strEnOceanSwitch_Rum_5_350B.bT2_OFF OR bBottomButtonZone1_Visu;
END_ACTION

ACTION A_LightCtrl:

fbLys(
	nZoneID:= 1, 
	bButtonZone1:= bTopButtonZone1,
	bBottomButtonZone1 := bBottomButtonZone1, 
	bButtonZone2:= bButtonZone2, 
	fLuxOn:= fLuxOn, 
	fLuxDim:= fLuxDim, 
	tPIRDim:= tPIRDim, 
	tPIROff:= tPIROff, 
	fOffsetSec:= fOffsetSec, 
	bReInit:= , 
	stDaliSetup:= stDaliSetup, 
	ipCommunication_Prim:= P_DALI_Background.arrfbKL6821Communication[DALI_LINE_NUM_LIGHT], 
	ipCommunication_Sec:= P_DALI_Background.arrfbKL6821Communication[DALI_LINE_NUM_LIGHT], 
	ipCommunication_Supl:= P_DALI_Background.arrfbKL6821Communication[DALI_LINE_NUM_LIGHT], 
	fMinOutputPowerLevelRoom:= 15, 
	fMaxOutputPowerLevelRoom:= 100, 
	nCycleTimeInMS:= 10 , 
	bRunTuning:= bRunTuning, 
	bOccupiedRoom=> bOccupiedRoom, 
	bError_Prim=> , 
	nError_Prim=> , 
	stTuneData:=stTuneData , 
	stPirSensorData:= stPirSensorData, 
	stLiveData:= stLiveData);
END_ACTION

ACTION A_Sensor:

fbSensor.ipCommunication := P_DALI_Background.arrfbKL6821Communication[Sensor_DALI_LINE_NUM];


fbSensor(
	byShrtAdr:= bySensorAddr,
	bInitialize:= bInitialize, 
	DALI_LINE_NUM:= Sensor_DALI_LINE_NUM, 
 	//bCancelHoldTimerOccupancy:= bCancelHoldTimerOccupancy, 
	stSensorSetup := stDaliSensorSetup,
	bInitErr=> bInitErr, 
	bInitDone=> bInitDone,
	stPirSensorData:= stPirSensorData, 
	arrSensorScales:= arrSensorScales);

(*
fbSensor(
	arrShrtAdr:= arrSensorAddr,
	bInitialize:= bInitialize, 
	DALI_LINE_NUM:= Sensor_DALI_LINE_NUM, 
 	//bCancelHoldTimerOccupancy:= bCancelHoldTimerOccupancy, 
	stSensorSetup := stDaliSensorSetup,
	arrInitErr=> arrInitErr, 
	arrInitDone=> arrInitDone,
	stPirSensorData:= stPirSensorData, 
	arrSensorScales:= arrSensorScales);
	*)
END_ACTION

END_PROGRAM

// ---- POUs/Alle_Rum/Rum_Med_DALI_Pir/Rum_5_350/P_Rum_5_350.TcPOU
PROGRAM P_Rum_5_350
VAR
//Light

	fbLys		: FB_Light_Type_A;
	
	stDaliSetup	: SH_Light.ST_DALI_RoomSetup := (		byShrtAdr_Prim := 43, 
														byGrpAdr_Prim := 10, 
														eMod_Prim := E_DALIAddressType.Group, 
														byShrtAdr_Sec := 1, 
														byGrpAdr_Sec := 1, 
														eMod_Sec := E_DALIAddressType.Short, 
														byShrtAdr_Supl := 1, 
														DALI_LINE_NUM_PRIM := DALI_LINE_NUM_LIGHT, 
														DALI_LINE_NUM_SEC := 0, //0 = ingen zonestyring/vinduerække
														DALI_LINE_NUM_SUPL := DALI_LINE_NUM_PENDANTS);
	stLiveData				: SH_Light.ST_LiveData;
	//stLiveData AT %MB22	: SH_Light.ST_LiveData;
	bTopButtonZone1			: BOOL;
	bTopButtonZone1_Visu	: BOOL;
	bBottomButtonZone1		: BOOL;
	bBottomButtonZone1_Visu	: BOOL;
	bButtonZone2			: BOOL;
	fLuxOn					: REAL := 500;
	fLuxDim					: REAL := 200;
	tPIRDim					: TIME := T#15M;
	tPIROff					: TIME := T#30M;
	fOffsetSec				: REAL := 20;
	bOccupiedRoom			: BOOL;

	bRunTuning				: BOOL;
	
// Sensor Settings
	fbSensor					: SH_Light.FB_NIKO_P46xx_1Pcs;
	//fbSensor					: SH_Light.FB_NIKO_P46xx_2Pcs;
	bySensorAddr				: BYTE := 15;
	//arrSensorAddr				: ARRAY[1..2] OF BYTE := [9,10];
	bInitialize					: BOOL := TRUE;
	stDaliSensorSetup			: ST_DALI_NIKOP46SetupData;
	bInitErr					: BOOL;
	bInitDone					: BOOL;
	//arrInitErr					: ARRAY [1..2] OF BOOL;
	//arrInitDone					: ARRAY [1..2] OF BOOL;
	arrSensorScales				: ARRAY [1..10] OF SH_Light.ST_DALI_SensorScaleMode := [	(fMeassureMaxSensor := 1023, fReadMaxSensor := 1023),
																						9(())];
	bCancelHoldTimerOccupancy	: BOOL;
(*	eEventPriorityOccupancy		: E_DALIEventPriority := E_DALIEVENTPRIORITY.Middle;
	nHoldTimerOccupancy			: WORD := 5; // Value in s. 	
	nReportTimerOccupancy		: BYTE := 120; // Value in s, Preset manufacturer value
	nDeadtimeTimerOccupancy		: WORD := 100; // Value in ms, Predefined Value of DALI Standard
	bCancelHoldTimerOccupancy	: BOOL;
	nSensitivityOccupancy		: BYTE:= 3; //setting Sensivity (0..4) 0 (Off), 1 (Min), 2(Low), 3(High) and 4 (Max)

	bEnableLuxEvent				: BOOL;
	eEventPriorityBrightness	: E_DALIEventPriority := E_DALIEVENTPRIORITY.Middle;
	nDeadtimeTimerBrightness	: WORD := 1500; // Value in ms, Predefined Value of DALI Standard
	nHysteresisBrightness		: BYTE := 2; // Value in %
	nHysteresisMinBrightness	: BYTE := 10; // Absolute Value, depending on the manufacturer specific resolution
	nReportTimerBrightness		: BYTE := 120; // Value in s, Preset manufacturer value
*)

END_VAR

VAR CONSTANT
	Sensor_DALI_LINE_NUM	: BYTE := 3;
	DALI_LINE_NUM_LIGHT		: BYTE := 1;
	DALI_LINE_NUM_PENDANTS	: BYTE := 0; //0=ingen pendler
END_VAR
VAR PERSISTENT
	stPirSensorData: SH_Light.ST_DALI_Sensor;
	stTuneData: SH_Light.ST_TuneData_EX;
END_VAR

A_Buttons();
A_LightCtrl();
A_Sensor();

ACTION A_Buttons:
bTopButtonZone1		:= GVL_EnOcean.strEnOceanSwitch_Rum_5_350.bT1_ON OR bTopButtonZone1_Visu;
bBottomButtonZone1	:= GVL_EnOcean.strEnOceanSwitch_Rum_5_350.bT1_OFF OR bBottomButtonZone1_Visu;
END_ACTION

ACTION A_LightCtrl:

fbLys(
	nZoneID:= 1, 
	bButtonZone1:= bTopButtonZone1,
	bBottomButtonZone1 := bBottomButtonZone1, 
	bButtonZone2:= bButtonZone2, 
	fLuxOn:= fLuxOn, 
	fLuxDim:= fLuxDim, 
	tPIRDim:= tPIRDim, 
	tPIROff:= tPIROff, 
	fOffsetSec:= fOffsetSec, 
	bReInit:= , 
	stDaliSetup:= stDaliSetup, 
	ipCommunication_Prim:= P_DALI_Background.arrfbKL6821Communication[DALI_LINE_NUM_LIGHT], 
	ipCommunication_Sec:= P_DALI_Background.arrfbKL6821Communication[DALI_LINE_NUM_LIGHT], 
	ipCommunication_Supl:= P_DALI_Background.arrfbKL6821Communication[DALI_LINE_NUM_LIGHT], 
	fMinOutputPowerLevelRoom:= 15, 
	fMaxOutputPowerLevelRoom:= 100, 
	nCycleTimeInMS:= 10 , 
	bRunTuning:= bRunTuning, 
	bOccupiedRoom=> bOccupiedRoom, 
	bError_Prim=> , 
	nError_Prim=> , 
	stTuneData:=stTuneData , 
	stPirSensorData:= stPirSensorData, 
	stLiveData:= stLiveData);
END_ACTION

ACTION A_Sensor:

fbSensor.ipCommunication := P_DALI_Background.arrfbKL6821Communication[Sensor_DALI_LINE_NUM];


fbSensor(
	byShrtAdr:= bySensorAddr,
	bInitialize:= bInitialize, 
	DALI_LINE_NUM:= Sensor_DALI_LINE_NUM, 
 	//bCancelHoldTimerOccupancy:= bCancelHoldTimerOccupancy, 
	stSensorSetup := stDaliSensorSetup,
	bInitErr=> bInitErr, 
	bInitDone=> bInitDone,
	stPirSensorData:= stPirSensorData, 
	arrSensorScales:= arrSensorScales);

(*
fbSensor(
	arrShrtAdr:= arrSensorAddr,
	bInitialize:= bInitialize, 
	DALI_LINE_NUM:= Sensor_DALI_LINE_NUM, 
 	//bCancelHoldTimerOccupancy:= bCancelHoldTimerOccupancy, 
	stSensorSetup := stDaliSensorSetup,
	arrInitErr=> arrInitErr, 
	arrInitDone=> arrInitDone,
	stPirSensorData:= stPirSensorData, 
	arrSensorScales:= arrSensorScales);
	*)
END_ACTION

END_PROGRAM

// ---- POUs/Alle_Rum/Rum_Med_DALI_Pir/Rum_5_355A_2tryk/P_Rum_5_355A.TcPOU
PROGRAM P_Rum_5_355A
VAR
//Light

	fbLys		: FB_Light_Type_A;
	
	stDaliSetup	: SH_Light.ST_DALI_RoomSetup := (		byShrtAdr_Prim := 30, 
														byGrpAdr_Prim := 6, 
														eMod_Prim := E_DALIAddressType.Group, 
														byShrtAdr_Sec := 1, 
														byGrpAdr_Sec := 1, 
														eMod_Sec := E_DALIAddressType.Short, 
														byShrtAdr_Supl := 1, 
														DALI_LINE_NUM_PRIM := DALI_LINE_NUM_LIGHT, 
														DALI_LINE_NUM_SEC := 0, //0 = ingen zonestyring/vinduerække
														DALI_LINE_NUM_SUPL := DALI_LINE_NUM_PENDANTS);
	stLiveData				: SH_Light.ST_LiveData;
	//stLiveData AT %MB22	: SH_Light.ST_LiveData;
	bTopButtonZone1			: BOOL;
	bTopButtonZone1_Visu	: BOOL;
	bBottomButtonZone1		: BOOL;
	bBottomButtonZone1_Visu	: BOOL;
	bButtonZone2			: BOOL;
	fLuxOn					: REAL := 500;
	fLuxDim					: REAL := 200;
	tPIRDim					: TIME := T#15M;
	tPIROff					: TIME := T#30M;
	fOffsetSec				: REAL := 20;
	bOccupiedRoom			: BOOL;

	bRunTuning				: BOOL;
	
// Sensor Settings
	fbSensor					: SH_Light.FB_NIKO_P46xx_1Pcs;
	//fbSensor					: SH_Light.FB_NIKO_P46xx_2Pcs;
	bySensorAddr				: BYTE := 7;
	//arrSensorAddr				: ARRAY[1..2] OF BYTE := [9,10];
	bInitialize					: BOOL := TRUE;
	stDaliSensorSetup			: ST_DALI_NIKOP46SetupData;
	bInitErr					: BOOL;
	bInitDone					: BOOL;
	//arrInitErr					: ARRAY [1..2] OF BOOL;
	//arrInitDone					: ARRAY [1..2] OF BOOL;
	arrSensorScales				: ARRAY [1..10] OF SH_Light.ST_DALI_SensorScaleMode := [	(fMeassureMaxSensor := 1023, fReadMaxSensor := 1023),
																						9(())];
	bCancelHoldTimerOccupancy	: BOOL;
(*	eEventPriorityOccupancy		: E_DALIEventPriority := E_DALIEVENTPRIORITY.Middle;
	nHoldTimerOccupancy			: WORD := 5; // Value in s. 	
	nReportTimerOccupancy		: BYTE := 120; // Value in s, Preset manufacturer value
	nDeadtimeTimerOccupancy		: WORD := 100; // Value in ms, Predefined Value of DALI Standard
	bCancelHoldTimerOccupancy	: BOOL;
	nSensitivityOccupancy		: BYTE:= 3; //setting Sensivity (0..4) 0 (Off), 1 (Min), 2(Low), 3(High) and 4 (Max)

	bEnableLuxEvent				: BOOL;
	eEventPriorityBrightness	: E_DALIEventPriority := E_DALIEVENTPRIORITY.Middle;
	nDeadtimeTimerBrightness	: WORD := 1500; // Value in ms, Predefined Value of DALI Standard
	nHysteresisBrightness		: BYTE := 2; // Value in %
	nHysteresisMinBrightness	: BYTE := 10; // Absolute Value, depending on the manufacturer specific resolution
	nReportTimerBrightness		: BYTE := 120; // Value in s, Preset manufacturer value
*)

END_VAR

VAR CONSTANT
	Sensor_DALI_LINE_NUM	: BYTE := 2;
	DALI_LINE_NUM_LIGHT		: BYTE := 1;
	DALI_LINE_NUM_PENDANTS	: BYTE := 0; //0=ingen pendler
END_VAR
VAR PERSISTENT
	stPirSensorData: SH_Light.ST_DALI_Sensor;
	stTuneData: SH_Light.ST_TuneData_EX;
END_VAR

A_Buttons();
A_LightCtrl();
A_Sensor();

ACTION A_Buttons:
bTopButtonZone1		:= GVL_EnOcean.strEnOceanSwitch_Rum_5_355A_Indgang1.bT1_OFF OR GVL_EnOcean.strEnOceanSwitch_Rum_5_355A_Indgang2.bT1_OFF OR bTopButtonZone1_Visu;
bBottomButtonZone1	:= GVL_EnOcean.strEnOceanSwitch_Rum_5_355A_Indgang1.bT1_ON OR GVL_EnOcean.strEnOceanSwitch_Rum_5_355A_Indgang2.bT1_ON OR bBottomButtonZone1_Visu;
END_ACTION

ACTION A_LightCtrl:

fbLys(
	nZoneID:= 1, 
	bButtonZone1:= bTopButtonZone1,
	bBottomButtonZone1 := bBottomButtonZone1, 
	bButtonZone2:= bButtonZone2, 
	fLuxOn:= fLuxOn, 
	fLuxDim:= fLuxDim, 
	tPIRDim:= tPIRDim, 
	tPIROff:= tPIROff, 
	fOffsetSec:= fOffsetSec, 
	bReInit:= , 
	stDaliSetup:= stDaliSetup, 
	ipCommunication_Prim:= P_DALI_Background.arrfbKL6821Communication[DALI_LINE_NUM_LIGHT], 
	ipCommunication_Sec:= P_DALI_Background.arrfbKL6821Communication[DALI_LINE_NUM_LIGHT], 
	ipCommunication_Supl:= P_DALI_Background.arrfbKL6821Communication[DALI_LINE_NUM_LIGHT], 
	fMinOutputPowerLevelRoom:= 15, 
	fMaxOutputPowerLevelRoom:= 100, 
	nCycleTimeInMS:= 10 , 
	bRunTuning:= bRunTuning, 
	bOccupiedRoom=> bOccupiedRoom, 
	bError_Prim=> , 
	nError_Prim=> , 
	stTuneData:=stTuneData , 
	stPirSensorData:= stPirSensorData, 
	stLiveData:= stLiveData);
END_ACTION

ACTION A_Sensor:

fbSensor.ipCommunication := P_DALI_Background.arrfbKL6821Communication[Sensor_DALI_LINE_NUM];


fbSensor(
	byShrtAdr:= bySensorAddr,
	bInitialize:= bInitialize, 
	DALI_LINE_NUM:= Sensor_DALI_LINE_NUM, 
 	//bCancelHoldTimerOccupancy:= bCancelHoldTimerOccupancy, 
	stSensorSetup := stDaliSensorSetup,
	bInitErr=> bInitErr, 
	bInitDone=> bInitDone,
	stPirSensorData:= stPirSensorData, 
	arrSensorScales:= arrSensorScales);

(*
fbSensor(
	arrShrtAdr:= arrSensorAddr,
	bInitialize:= bInitialize, 
	DALI_LINE_NUM:= Sensor_DALI_LINE_NUM, 
 	//bCancelHoldTimerOccupancy:= bCancelHoldTimerOccupancy, 
	stSensorSetup := stDaliSensorSetup,
	arrInitErr=> arrInitErr, 
	arrInitDone=> arrInitDone,
	stPirSensorData:= stPirSensorData, 
	arrSensorScales:= arrSensorScales);
	*)
END_ACTION

END_PROGRAM

// ---- POUs/Alle_Rum/Trapper/P_Trappe.TcPOU
PROGRAM P_Trappe
VAR
	
	
	DigIn3	AT %I* :	BOOL;
	DigIn4	AT %I* :	BOOL;
	DigIn5	AT %I* :	BOOL;
	DigIn6	AT %I* :	BOOL;
	DigIn7	AT %I* :	BOOL;
	DigIn8	AT %I* :	BOOL;
	
	DigOut1 AT %Q*	:	BOOL;
END_VAR

END_PROGRAM

// ---- POUs/DALI/DALI_Setup/FBs/FB_Part102Commands.TcPOU
FUNCTION_BLOCK FB_Part102Commands
VAR_INPUT
	ipDALICommunication		:	I_DALICommunication;
END_VAR
VAR_OUTPUT
	bBusy					:	BOOL;
END_VAR
VAR
	{region "Visu"}
	eAddressType			:	E_DALIAddressType;
	nShortAddress			:	BYTE := 255;
	nGroupAddress			:	BYTE := 255;
	bRecallMaxLevel			:	BOOL;
	bRecallMinLevel			:	BOOL;
	bOff					:	BOOL;
	bUp						:	BOOL;
	bStepUp					:	BOOL;
	bOnAndStepUp			:	BOOL;
	bStepDownAndOff			:	BOOL;
	bDown					:	BOOL;
	bStepDown				:	BOOL;
	bGotoScene				:	BOOL;
	nScene					:	BYTE;
	sActualLevel			:	STRING(5);
	sControlGearFailure		:	STRING(5);
	sLampFailure			:	STRING(5);
	sFadeRunning			:	STRING(5);
	sResetState				:	STRING(5);
	{endregion}
	nStep					:	INT;
	nStepQuery				:	INT;
	tonDelay				:	TON;
	nAddress				:	BYTE := 255;
	fbRecallMaxLevel		:	FB_DALI102RecallMaxLevel(0);
	fbRecallMinLevel		:	FB_DALI102RecallMinLevel(0);
	fbOff					:	FB_DALI102Off(0);
	fbUp					:	FB_DALI102Up(0);
	fbStepUp				:	FB_DALI102StepUp(0);
	fbOnAndStepUp			:	FB_DALI102OnAndStepUp(0);
	fbStepDownAndOff		:	FB_DALI102StepDownAndOff(0);
	fbDown					:	FB_DALI102Down(0);
	fbStepDown				:	FB_DALI102StepDown(0);
	fbGotoScene				:	FB_DALI102GotoScene(0);
	fbQueryActualLevel		:	FB_DALI102QueryActualLevel(0);
	fbQueryStatus			:	FB_DALI102QueryStatus(0);
END_VAR

{region "Detect Commands"}
IF (bRecallMaxLevel AND (nStep = 0)) THEN
	nStep := 10;
	bRecallMaxLevel := FALSE;
END_IF

IF (bRecallMinLevel AND (nStep = 0)) THEN
	nStep := 20;
	bRecallMinLevel := FALSE;
END_IF

IF (bOff AND (nStep = 0)) THEN
	nStep := 30;
	bOff := FALSE;
END_IF

IF (bUp AND (nStep = 0)) THEN
	nStep := 40;
	bUp := FALSE;
END_IF

IF (bStepUp AND (nStep = 0)) THEN
	nStep := 50;
	bStepUp := FALSE;
END_IF

IF (bOnAndStepUp AND (nStep = 0)) THEN
	nStep := 60;
	bOnAndStepUp := FALSE;
END_IF

IF (bStepDownAndOff AND (nStep = 0)) THEN
	nStep := 70;
	bStepDownAndOff := FALSE;
END_IF

IF (bDown AND (nStep = 0)) THEN
	nStep := 80;
	bDown := FALSE;
END_IF

IF (bStepDown AND (nStep = 0)) THEN
	nStep := 90;
	bStepDown := FALSE;
END_IF

IF (bGotoScene AND (nStep = 0)) THEN
	nStep := 100;
	bGotoScene := FALSE;
END_IF
{endregion}
{region "Manage Dialog Selection}
IF (nStep = 0) THEN
	bBusy := FALSE;
ELSE
	bBusy := TRUE;
END_IF
{endregion}
{region "Execute Commands"}
nAddress := SEL(eAddressType = E_DALIAddressType.Short, nGroupAddress, nShortAddress);
CASE nStep OF
0:
{region "Init"}
	bRecallMaxLevel := FALSE;
	bRecallMinLevel := FALSE;
	bOff := FALSE;
	bUp := FALSE;
	bStepUp := FALSE;
	bOnAndStepUp := FALSE;
	bStepDownAndOff := FALSE;
	bDown := FALSE;
	bStepDown := FALSE;
	bGotoScene := FALSE;

	fbRecallMaxLevel.ipDALICommunication := ipDALICommunication;
	fbRecallMinLevel.ipDALICommunication := ipDALICommunication;
	fbOff.ipDALICommunication := ipDALICommunication;
	fbUp.ipDALICommunication := ipDALICommunication;
	fbStepUp.ipDALICommunication := ipDALICommunication;
	fbOnAndStepUp.ipDALICommunication := ipDALICommunication;
	fbStepDownAndOff.ipDALICommunication := ipDALICommunication;
	fbDown.ipDALICommunication := ipDALICommunication;
	fbStepDown.ipDALICommunication := ipDALICommunication;
	fbGotoScene.ipDALICommunication := ipDALICommunication;
	fbQueryActualLevel.ipDALICommunication := ipDALICommunication;
	fbQueryStatus.ipDALICommunication := ipDALICommunication;
{endregion}
10:
{region "Recall Max Level"}
	fbRecallMaxLevel(bStart := TRUE,
					 nAddress := nAddress,
					 eAddressType := eAddressType,
					 eCommandPriority := E_DALICommandPriority.Middle);
	IF (NOT fbRecallMaxLevel.bBusy) THEN
		fbRecallMaxLevel(bStart := FALSE);
		nStep := 0;
	END_IF
{endregion}
20:
{region "Recall Min Level"}
	fbRecallMinLevel(bStart := TRUE,
					 nAddress := nAddress,
					 eAddressType := eAddressType,
					 eCommandPriority := E_DALICommandPriority.Middle);
	IF (NOT fbRecallMinLevel.bBusy) THEN
		fbRecallMinLevel(bStart := FALSE);
		nStep := 0;
	END_IF
{endregion}
30:
{region "Off"}
	fbOff(bStart := TRUE,
		  nAddress := nAddress,
		  eAddressType := eAddressType,
		  eCommandPriority := E_DALICommandPriority.Middle);
	IF (NOT fbOff.bBusy) THEN
		fbOff(bStart := FALSE);
		nStep := 0;
	END_IF
{endregion}
40:
{region "Up"}
	fbUp(bStart := TRUE,
		 nAddress := nAddress,
		 eAddressType := eAddressType,
		 eCommandPriority := E_DALICommandPriority.Middle);
	IF (NOT fbUp.bBusy) THEN
		fbUp(bStart := FALSE);
		nStep := 0;
	END_IF
{endregion}
50:
{region "Step Up"}
	fbStepUp(bStart := TRUE,
			 nAddress := nAddress,
			 eAddressType := eAddressType,
			 eCommandPriority := E_DALICommandPriority.Middle);
	IF (NOT fbStepUp.bBusy) THEN
		fbStepUp(bStart := FALSE);
		nStep := 0;
	END_IF
{endregion}
60:
{region "On and Step Up"}
	fbOnAndStepUp(	bStart := TRUE,
					nAddress := nAddress,
					eAddressType := eAddressType,
					eCommandPriority := E_DALICommandPriority.Middle);
	IF (NOT fbOnAndStepUp.bBusy) THEN
		fbOnAndStepUp(bStart := FALSE);
		nStep := 0;
	END_IF
{endregion}
70:
{region "Step Down and Step Off"}
	fbStepDownAndOff(	bStart := TRUE,
						nAddress := nAddress,
						eAddressType := eAddressType,
						eCommandPriority := E_DALICommandPriority.Middle);
	IF (NOT fbStepDownAndOff.bBusy) THEN
		fbStepDownAndOff(bStart := FALSE);
		nStep := 0;
	END_IF
{endregion}
80:
{region "Down"}
	fbDown(	bStart := TRUE,
			nAddress := nAddress,
			eAddressType := eAddressType,
			eCommandPriority := E_DALICommandPriority.Middle);
	IF (NOT fbDown.bBusy) THEN
		fbDown(bStart := FALSE);
		nStep := 0;
	END_IF
{endregion}
90:
{region "Step Down"}
	fbStepDown(	bStart := TRUE,
				nAddress := nAddress,
				eAddressType := eAddressType,
				eCommandPriority := E_DALICommandPriority.Middle);
	IF (NOT fbStepDown.bBusy) THEN
		fbStepDown(bStart := FALSE);
		nStep := 0;
	END_IF
{endregion}
100:
{region "Goto Scene"}
	fbGotoScene(bStart := TRUE,
				nAddress := nAddress,
				eAddressType := eAddressType,
				eCommandPriority := E_DALICommandPriority.Middle,
				nScene := nScene);
	IF (NOT fbGotoScene.bBusy) THEN
		fbGotoScene(bStart := FALSE);
		nStep := 0;
	END_IF
{endregion}
ELSE
	nStep := 0;
END_CASE
{endregion}

{region "Query Actual Level / Query Status"}
CASE nStepQuery OF
0:
	tonDelay(IN := TRUE, PT := T#1S);
	IF (tonDelay.Q) THEN
		tonDelay(IN := FALSE);
		IF ((nAddress <> 255) AND (eAddressType = E_DALIAddressType.Short)) THEN
			nStepQuery := 10;
		ELSE
			sActualLevel := '???';
			sControlGearFailure := '???';
			sLampFailure := '???';
			sFadeRunning := '???';
			sResetState := '???';
		END_IF
	END_IF
10:
	fbQueryActualLevel(	bStart := TRUE,
						nAddress := nAddress,
						eAddressType := eAddressType,
						eCommandPriority := E_DALICommandPriority.Middle);
	IF (NOT fbQueryActualLevel.bBusy) THEN
		IF (NOT fbQueryActualLevel.bError) THEN
			sActualLevel := TO_STRING(fbQueryActualLevel.nActualLevel);
		ELSE
			sActualLevel := '???';
		END_IF
		fbQueryActualLevel(bStart := FALSE);
		nStepQuery := 20;
	END_IF
20:
	fbQueryStatus(	bStart := TRUE,
					nAddress := nAddress,
					eAddressType := eAddressType,
					eCommandPriority := E_DALICommandPriority.Middle);
	IF (NOT fbQueryStatus.bBusy) THEN
		IF (NOT fbQueryStatus.bError) THEN
			sControlGearFailure := SEL(fbQueryStatus.nStatus.0, 'False', 'True');
			sLampFailure := SEL(fbQueryStatus.nStatus.1, 'False', 'True');
			sFadeRunning := SEL(fbQueryStatus.nStatus.4, 'False', 'True');
			sResetState := SEL(fbQueryStatus.nStatus.5, 'False', 'True');
		ELSE
			sControlGearFailure := '???';
			sLampFailure := '???';
			sFadeRunning := '???';
			sResetState := '???';
		END_IF
		fbQueryStatus(bStart := FALSE);
		nStepQuery := 0;
	END_IF

ELSE
	nStepQuery := 0;
END_CASE
{endregion}

END_FUNCTION_BLOCK

// ---- POUs/DALI/DALI_Setup/FBs/FB_Part102Scenes.TcPOU
FUNCTION_BLOCK FB_Part102Scenes
VAR_INPUT
	ipDALICommunication		:	I_DALICommunication;
END_VAR
VAR_OUTPUT
	bBusy					:	BOOL;
END_VAR
VAR
	{region "Visu"}
	nScene					:	BYTE;
	bGoToScene				:	BOOL;
	bSwitchOff				:	BOOL;
	bRead					:	BOOL;
	bWrite		 			:	BOOL;
	aScene					:	ARRAY [0..63] OF BYTE;
	aNoShortAddress			:	ARRAY [0..63] OF BOOL;
	bHideWaitSymbol			:	BOOL := TRUE;
	{endregion}
	nStep					:	INT; // Running index
	nAddress				:	INT;
	aFont					:	ARRAY [0..63] OF DWORD;

	fb103StartQuiescentMode	:	FB_DALI103StartQuiescentMode(0);
	fb103StopQuiescentMode	:	FB_DALI103StopQuiescentMode(0);
	fb102QuerySceneLevel	:	FB_DALI102QuerySceneLevel(0);
	fb102SetScene			:	FB_DALI102SetScene(0);
	fb102GoToScene			:	FB_DALI102GoToScene(0);
	fb102Off				:	FB_DALI102Off(0);
END_VAR

{region "Detect Commands"}
IF (bRead AND (nStep = 0)) THEN 
	nStep := 5;
	bRead := FALSE;
	bHideWaitSymbol := FALSE;
END_IF

IF (bWrite AND (nStep = 0)) THEN 
	nStep := 20;
	bWrite := FALSE;
	bHideWaitSymbol := FALSE;
END_IF

IF (bGoToScene AND (nStep = 0)) THEN 
	nStep := 30;
	bGoToScene := FALSE;
	bHideWaitSymbol := FALSE;
END_IF

IF (bSwitchOff AND (nStep = 0)) THEN
	nStep := 40;
	bSwitchOff := FALSE;
	bHideWaitSymbol := FALSE;
END_IF
{endregion}
{region "Manage Dialog Selection}
IF (nStep = 0) THEN
	bBusy := FALSE;
ELSE
	bBusy := TRUE;
END_IF
{endregion}
{region "Execute Commands"}
CASE nStep OF
0:
{region "Init"}
	bRead := FALSE;	
	bWrite := FALSE;
	bGoToScene := FALSE;
	bSwitchOff := FALSE;
	bHideWaitSymbol := TRUE;
	nAddress := 0;

	fb103StartQuiescentMode.ipDALICommunication := ipDALICommunication;
	fb103StopQuiescentMode.ipDALICommunication := ipDALICommunication;
	fb102QuerySceneLevel.ipDALICommunication := ipDALICommunication;
	fb102SetScene.ipDALICommunication := ipDALICommunication;
	fb102GoToScene.ipDALICommunication := ipDALICommunication;
	fb102Off.ipDALICommunication := ipDALICommunication;
{endregion}
5:
{region "Start Qiescent Mode"}
	fb103StartQuiescentMode(bStart := TRUE,
							eAddressType := Tc3_DALI.E_DALIAddressType.Broadcast,
							eCommandPriority := Tc3_DALI.E_DALICommandPriority.Middle);
	IF (NOT fb103StartQuiescentMode.bBusy) THEN
		fb103StartQuiescentMode(bStart:= FALSE);
		nStep := 10;
	END_IF
{endregion}
10:
{region "Query Scene Level"}
	fb102QuerySceneLevel(	bStart := TRUE,
							nAddress := TO_BYTE(nAddress),
							eAddressType := Tc3_DALI.E_DALIAddressType.Short,
							eCommandPriority := Tc3_DALI.E_DALICommandPriority.Middle,
							nScene := nScene,
							nSceneLevel=> aScene[nAddress]);
	IF (NOT fb102QuerySceneLevel.bBusy) THEN
		fb102QuerySceneLevel (bStart:= FALSE);
		IF (fb102QuerySceneLevel.ipResultMessage.nEventId = TC_EVENTS.TcDALIEventClass.NoResponseFromTheDALIDevice.nEventId) THEN // Deletes not existing short addresses from display
			aNoShortAddress[nAddress] := TRUE;
			aFont[nAddress] := 16#FF505050;
		ELSE
			aNoShortAddress[nAddress] := FALSE;
			aFont[nAddress] := 16#FFFFFFFF;
		END_IF
		nAddress := nAddress + 1;
		IF (nAddress > 63)THEN
			nStep := 15;
		END_IF
	END_IF
{endregion}
15:
{region "Stop Qiescent Mode"}
	fb103StopQuiescentMode(	bStart := TRUE,
							eAddressType := Tc3_DALI.E_DALIAddressType.Broadcast,
							eCommandPriority := Tc3_DALI.E_DALICommandPriority.Middle);
	IF (NOT fb103StopQuiescentMode.bBusy) THEN
		fb103StopQuiescentMode(	bStart:= FALSE);
		nStep := 0;
	END_IF
{endregion}
20:
{region "Set Scene"}
	IF (aNoShortAddress[nAddress] = TRUE) THEN
		nAddress := nAddress + 1;
		IF (nAddress > 63)THEN
			nStep := 0;
		END_IF
	ELSE
		fb102SetScene(	bStart := TRUE,
						nAddress := TO_BYTE(nAddress),
						eAddressType := Tc3_DALI.E_DALIAddressType.Short,
						eCommandPriority := Tc3_DALI.E_DALICommandPriority.Middle,
						nSceneLevel := aScene[nAddress],
						nScene := nScene);
		IF (NOT fb102SetScene.bBusy) THEN
			fb102SetScene(bStart := FALSE);
			nAddress := nAddress + 1;
			IF (nAddress > 63)THEN
				nStep := 0;
			END_IF
		END_IF
	END_IF
{endregion}
30:
{region "Go To Scene"}
	IF (aNoShortAddress[nAddress] = TRUE) THEN
		nAddress := nAddress + 1;
		IF (nAddress > 63)THEN
			nStep := 0;
		END_IF
	ELSE
		fb102GoToScene(	bStart := TRUE,
						nAddress := TO_BYTE(nAddress),
						eAddressType := Tc3_DALI.E_DALIAddressType.Short,
						eCommandPriority := Tc3_DALI.E_DALICommandPriority.Middle,
						nScene := nScene);
		IF (NOT fb102GoToScene.bBusy) THEN
			fb102GoToScene(bStart := FALSE);
			nAddress := nAddress + 1;
			IF (nAddress > 63)THEN
				nStep := 0;
			END_IF
		END_IF
	END_IF
{endregion}
40:
{region "Switch Off"}
	fb102Off(	bStart := TRUE,
				nAddress := TO_BYTE(nAddress),
				eAddressType := Tc3_DALI.E_DALIAddressType.Broadcast,
				eCommandPriority := Tc3_DALI.E_DALICommandPriority.Middle);
	IF (NOT fb102Off.bBusy) THEN
		fb102Off(bStart := FALSE);
		nStep := 0;
	END_IF
{endregion}
END_CASE
{endregion}

END_FUNCTION_BLOCK

// ---- POUs/DALI/DALI_Setup/FBs/FB_Part202Emergency.TcPOU
FUNCTION_BLOCK FB_Part202Emergency
VAR_INPUT
	ipDALICommunication					:	I_DALICommunication;
END_VAR
VAR_OUTPUT
	bBusy								:	BOOL;
END_VAR
VAR
	{region "Visu"}
	bReadCommands						:	BOOL;
	bReadState							:	BOOL;
	bReadParameter						:	BOOL;
	bStartFunctionTest					:	BOOL;
	bStopTest							:	BOOL;
	bStartDurationTest					:	BOOL;
	bResetFunctionTestDoneFlag			:	BOOL;
	bResetDurationTestDoneFlag			:	BOOL;
	bInhibit							:	BOOL;
	bResetInhibit						:	BOOL;
	bResetLampTime						:	BOOL;
	bRest								:	BOOL;
	bStartIdentification				:	BOOL;
	bWrite								:	BOOL;
	nBatteryCharge						:	BYTE;
	nDurationTestResult					:	BYTE;
	nLampEmergencyTime					:	BYTE;
	nLampTotalOperationTime				:	BYTE;
	sRestMode							:	STRING[5];
	sNormalMode							:	STRING[5];
	sEmergencyMode						:	STRING[5];
	sExtendedEmergency					:	STRING[5];
	sFunctionTest						:	STRING[5];
	sDurationTest						:	STRING[5];
	sHardwiredInhibit					:	STRING[5];
	sHardwiredSwitch					:	STRING[5];

	sCircuitFailure						:	STRING[5];
	sBatteryDurationFailure				:	STRING[5];
	sBatteryFailure						:	STRING[5];
	sEmergencyLampFailure				:	STRING[5];
	sFunctionTestExceed					:	STRING[5];
	sDurationTestExceed					:	STRING[5];
	sFunctionTestFailed					:	STRING[5];
	sDurationTestFailed					:	STRING[5];

	sInhibitMode						:	STRING[5];
	sFunctionTestDoneValid				:	STRING[5];
	sDurationTestDoneValid				:	STRING[5];
	sBatteryFullCharged					:	STRING[5];
	sFunctionTestRequestPending			:	STRING[5];
	sDurationTestRequestPending			:	STRING[5];
	sIdentificationActive				:	STRING[5];

	bIntegralControlGear				:	BOOL;
	bMaintainedControlGear				:	BOOL;
	bSwitchtedMaintainedControlGear		:	BOOL;
	bAutoTestCapability					:	BOOL;
	bAdjustableEmergencyLevel			:	BOOL;
	bHardwiredInhibitSupported			:	BOOL;
	bPhysicalSelectionSupported			:	BOOL;
	bRelightinRestModeSupported			:	BOOL;

	nEmergencyLevel						:	BYTE;
	nEmergencyMinLevel					:	BYTE;
	nEmergencyMaxLevel					:	BYTE;
	nProlongTime						:	UINT;
	fDurationTestDelayTimeVisu			:	REAL;
	fFunctionTestDelayTimeVisu			:	REAL;
	nFunctionTestInterval				:	UINT;
	nDurationTestInterval				:	UINT;
	nTestExecutionTimeout				:	UINT;
	nRatedDuration						:	BYTE;
	{endregion}
	nStep								:	INT;
	nAddress							:	BYTE;
	bHideWaitSymbol						:	BOOL := TRUE;
	
	nDurationTestDelayTime				:	UINT;
	nFunctionTestDelayTime				:	UINT;
	
	fb103StartQuiescentMode				:	FB_DALI103StartQuiescentMode(0);
	fb103StopQuiescentMode				:	FB_DALI103StopQuiescentMode(0);
	fb202QueryBatteryCharge				:	FB_DALI202QueryBatteryCharge(0);
	fb202QueryDurationTestResult		:	FB_DALI202QueryDurationTestResult(0);
	fb202QueryLampEmergencyTime			:	FB_DALI202QueryLampEmergencyTime(0);
	fb202QueryLampTotalOperationTime	:	FB_DALI202QueryLampTotalOperationTime(0);
	fb202QueryEmergencyLevel			:	FB_DALI202QueryEmergencyLevel(0);
	fb202QueryEmergencyMode				:	FB_DALI202QueryEmergencyMode(0);
	fb202QueryFailureStatus				:	FB_DALI202QueryFailureStatus(0);
	fb202QueryEmergencyStatus			:	FB_DALI202QueryEmergencyStatus(0);
	
	fb202QueryEmergencyMinLevel			:	FB_DALI202QueryEmergencyMinLevel(0);
	fb202QueryEmergencyMaxLevel			:	FB_DALI202QueryEmergencyMaxLevel(0);
	fb202QueryTestTiming				:	FB_DALI202QueryTestTiming(0);
	fb202QueryRatedDuration				:	FB_DALI202QueryRatedDuration(0);
	fb202QueryFeatures					:	FB_DALI202QueryFeatures(0);
	
	fb202SetEmergencyLevel				:	FB_DALI202SetEmergencyLevel(0);
	fb202SetProlongTime					:	FB_DALI202SetProlongTime(0);
	fb202SetTestDelayTime				:	FB_DALI202SetTestDelayTime(0);
	fb202SetFunctionTestInterval		:	FB_DALI202SetFunctionTestInterval(0);
	fb202SetDurationTestInterval		:	FB_DALI202SetDurationTestInterval(0);
	fb202SetTestExecutionTimeout		:	FB_DALI202SetTestExecutionTimeout(0);
	
	fb202StartFunctionTest				:	FB_DALI202StartFunctionTest(0);
	fb202StopTest						:	FB_DALI202StopTest(0);
	fb202StartDurationTest				:	FB_DALI202StartDurationTest(0);
	fb202ResetFunctionTestDoneFlag		:	FB_DALI202ResetFunctionTestDoneFlag(0);
	fb202ResetDurationTestDoneFlag		:	FB_DALI202ResetDurationTestDoneFlag(0);
	fb202Inhibit						:	FB_DALI202Inhibit(0);
	fb202ReLightResetInhibit			:	FB_DALI202ReLightResetInhibit(0);
	fb202ResetLampTime					:	FB_DALI202ResetLampTime(0);
	fb202Rest							:	FB_DALI202Rest(0);
	fb202StartIdentification			:	FB_DALI202StartIdentification(0);
END_VAR

{region "Detect Commands"}
IF (bStartFunctionTest AND (nStep = 0)) THEN
	nStep := 5;
	bStartFunctionTest := FALSE;
END_IF

IF (bStopTest AND (nStep = 0)) THEN
	nStep := 10;
	bStopTest := FALSE;
END_IF

IF (bStartDurationTest AND (nStep = 0)) THEN
	nStep := 15;
	bStartDurationTest := FALSE;
END_IF

IF (bResetFunctionTestDoneFlag AND (nStep = 0)) THEN
	nStep := 20;
	bResetFunctionTestDoneFlag := FALSE;
END_IF

IF (bResetDurationTestDoneFlag AND (nStep = 0)) THEN
	nStep := 25;
	bResetDurationTestDoneFlag := FALSE;
END_IF

IF (bInhibit AND (nStep = 0)) THEN
	nStep := 30;
	bInhibit := FALSE;
END_IF

IF (bResetInhibit AND (nStep = 0)) THEN
	nStep := 35;
	bResetInhibit := FALSE;
END_IF

IF (bResetLampTime AND (nStep = 0)) THEN
	nStep := 40;
	bResetLampTime := FALSE;
END_IF			   
					
IF (bRest AND (nStep = 0)) THEN
	nStep := 45;
	bRest := FALSE;
END_IF

IF (bStartIdentification AND (nStep = 0)) THEN
	nStep := 50;
	bStartIdentification := FALSE;
END_IF

IF (bReadCommands AND (nStep = 0)) THEN
	nStep := 60;
	bReadCommands := FALSE;
	bHideWaitSymbol := FALSE;
END_IF

IF (bReadState AND (nStep = 0)) THEN
	nStep := 100;
	bReadState := FALSE;
	bHideWaitSymbol := FALSE;
END_IF

IF (bReadParameter AND (nStep = 0)) THEN
	nStep := 200;
	bReadParameter := FALSE;
	bHideWaitSymbol := FALSE;
END_IF

IF (bWrite AND (nStep = 0)) THEN
	nStep := 500;
	bWrite := FALSE;
	bHideWaitSymbol := FALSE;
END_IF
{endregion}
{region "Manage Dialog Selection}
IF (nStep = 0) THEN
	bBusy := FALSE;
ELSE
	bBusy := TRUE;
END_IF
{endregion}
{region "Execute Commands"}
CASE nStep OF
0:
{region "Init"}
	bReadCommands := FALSE;
	bReadState := FALSE;
	bReadParameter := FALSE;
	bWrite := FALSE;
	bHideWaitSymbol := TRUE;

	fb103StartQuiescentMode.ipDALICommunication := ipDALICommunication;
	fb103StopQuiescentMode.ipDALICommunication := ipDALICommunication;
	fb202QueryBatteryCharge.ipDALICommunication := ipDALICommunication;
	fb202QueryDurationTestResult.ipDALICommunication := ipDALICommunication;
	fb202QueryDurationTestResult.ipDALICommunication := ipDALICommunication;
	fb202QueryLampEmergencyTime.ipDALICommunication := ipDALICommunication;
	fb202QueryLampTotalOperationTime.ipDALICommunication := ipDALICommunication;
	fb202QueryEmergencyMode.ipDALICommunication := ipDALICommunication;
	fb202QueryFailureStatus.ipDALICommunication := ipDALICommunication;
	fb202QueryEmergencyStatus.ipDALICommunication := ipDALICommunication;
	fb202QueryEmergencyLevel.ipDALICommunication := ipDALICommunication;
	fb202QueryEmergencyMinLevel.ipDALICommunication := ipDALICommunication;
	fb202QueryEmergencyMaxLevel.ipDALICommunication := ipDALICommunication;
	fb202QueryTestTiming.ipDALICommunication := ipDALICommunication;
	fb202QueryRatedDuration.ipDALICommunication := ipDALICommunication;
	fb202QueryFeatures.ipDALICommunication := ipDALICommunication;
	fb202SetEmergencyLevel.ipDALICommunication := ipDALICommunication;
	fb202SetProlongTime.ipDALICommunication := ipDALICommunication;
	fb202SetTestDelayTime.ipDALICommunication := ipDALICommunication;
	fb202SetFunctionTestInterval.ipDALICommunication := ipDALICommunication;
	fb202SetDurationTestInterval.ipDALICommunication := ipDALICommunication;
	fb202SetTestExecutionTimeout.ipDALICommunication := ipDALICommunication;

	fb202StartFunctionTest.ipDALICommunication := ipDALICommunication;
	fb202StopTest.ipDALICommunication := ipDALICommunication;
	fb202StartDurationTest.ipDALICommunication := ipDALICommunication;
	fb202ResetFunctionTestDoneFlag.ipDALICommunication := ipDALICommunication;
	fb202ResetDurationTestDoneFlag.ipDALICommunication := ipDALICommunication;
	fb202Inhibit.ipDALICommunication := ipDALICommunication;
	fb202ReLightResetInhibit.ipDALICommunication := ipDALICommunication;
	fb202ResetLampTime.ipDALICommunication := ipDALICommunication;
	fb202Rest.ipDALICommunication := ipDALICommunication;
	fb202StartIdentification.ipDALICommunication := ipDALICommunication;
{endregion}
{region "Commands"}
5:
	fb202StartFunctionTest(	bStart:= TRUE,
							nAddress := nAddress,
							eAddressType := Tc3_DALI.E_DALIAddressType.Short,
							eCommandPriority := Tc3_DALI.E_DALICommandPriority.Middle);
	IF (NOT fb202StartFunctionTest.bBusy) THEN
		fb202StartFunctionTest(bStart := FALSE);
		nStep :=0;
	END_IF
10:
	fb202StopTest(	bStart:= TRUE,
					nAddress := nAddress,
					eAddressType := Tc3_DALI.E_DALIAddressType.Short,
					eCommandPriority := Tc3_DALI.E_DALICommandPriority.Middle);
	IF (NOT fb202StopTest.bBusy) THEN
		fb202StopTest(bStart := FALSE);
		nStep :=0;
	END_IF
15:
	fb202StartDurationTest(	bStart:= TRUE,
							nAddress := nAddress,
							eAddressType := Tc3_DALI.E_DALIAddressType.Short,
							eCommandPriority := Tc3_DALI.E_DALICommandPriority.Middle);
	IF (NOT fb202StartDurationTest.bBusy) THEN
		fb202StartDurationTest(bStart := FALSE);
		nStep := 0;
	END_IF
20:
	fb202ResetFunctionTestDoneFlag(	bStart := TRUE,
									nAddress := nAddress,
									eAddressType := Tc3_DALI.E_DALIAddressType.Short,
									eCommandPriority := Tc3_DALI.E_DALICommandPriority.Middle);
	IF (NOT fb202ResetFunctionTestDoneFlag.bBusy) THEN
		fb202ResetFunctionTestDoneFlag(bStart := FALSE);
		nStep := 0;
	END_IF
25:
	fb202ResetDurationTestDoneFlag(	bStart:= TRUE,
									nAddress := nAddress,
									eAddressType := Tc3_DALI.E_DALIAddressType.Short,
									eCommandPriority := Tc3_DALI.E_DALICommandPriority.Middle);
	IF (NOT fb202ResetDurationTestDoneFlag.bBusy) THEN
		fb202ResetDurationTestDoneFlag(bStart := FALSE);
		nStep := 0;
	END_IF
30:
	fb202Inhibit(	bStart := TRUE,
					nAddress := nAddress,
					eAddressType := Tc3_DALI.E_DALIAddressType.Short,
					eCommandPriority := Tc3_DALI.E_DALICommandPriority.Middle);
	IF (NOT fb202Inhibit.bBusy) THEN
		fb202Inhibit(bStart := FALSE);
		nStep := 0;
	END_IF
35:
	fb202ReLightResetInhibit(	bStart := TRUE,
								nAddress := nAddress,
								eAddressType := Tc3_DALI.E_DALIAddressType.Short,
								eCommandPriority := Tc3_DALI.E_DALICommandPriority.Middle);
	IF (NOT fb202ReLightResetInhibit.bBusy) THEN
		fb202ReLightResetInhibit(bStart := FALSE);
		nStep := 0;
	END_IF
40:
	fb202ResetLampTime(	bStart := TRUE,
						nAddress := nAddress,
						eAddressType := Tc3_DALI.E_DALIAddressType.Short,
						eCommandPriority := Tc3_DALI.E_DALICommandPriority.Middle);
	IF (NOT fb202ResetLampTime.bBusy) THEN
		fb202ResetLampTime(bStart := FALSE);
		nStep := 0;
	END_IF
45:
	fb202Rest(	bStart := TRUE,
				nAddress := nAddress,
				eAddressType := Tc3_DALI.E_DALIAddressType.Short,
				eCommandPriority := Tc3_DALI.E_DALICommandPriority.Middle);
	IF (NOT fb202Rest.bBusy) THEN
		fb202Rest(bStart := FALSE);
		nStep := 0;
	END_IF
50:
	fb202StartIdentification(	bStart := TRUE,
								nAddress := nAddress,
								eAddressType := Tc3_DALI.E_DALIAddressType.Short,
								eCommandPriority := Tc3_DALI.E_DALICommandPriority.Middle);
	IF (NOT fb202StartIdentification.bBusy) THEN
		fb202StartIdentification(bStart := FALSE);
		nStep := 0;
	END_IF
{endregion}
{region "Read Command Status"}
55:
{region "Start Qiescent Mode"}
	fb103StartQuiescentMode(bStart := TRUE,
							eAddressType := Tc3_DALI.E_DALIAddressType.Broadcast,
							eCommandPriority := Tc3_DALI.E_DALICommandPriority.Middle);
	IF (NOT fb103StartQuiescentMode.bBusy) THEN
		fb103StartQuiescentMode(bStart := FALSE);
		nStep := 60;
	END_IF
{endregion}
{endregion}
60:
{region "Query Battery Charge"}
	fb202QueryBatteryCharge(bStart := TRUE,
							nAddress := nAddress,
							eAddressType := Tc3_DALI.E_DALIAddressType.Short,
							eCommandPriority := Tc3_DALI.E_DALICommandPriority.Middle );
	IF (NOT fb202QueryBatteryCharge.bBusy) THEN
		fb202QueryBatteryCharge(bStart:= FALSE);
		nBatteryCharge := fb202QueryBatteryCharge.nBatteryCharge;
		nStep := 65;
	END_IF
{endregion}
65:
{region "Query Duration Test Result"}
	fb202QueryDurationTestResult(	bStart := TRUE,
									nAddress := nAddress,
									eAddressType := Tc3_DALI.E_DALIAddressType.Short,
									eCommandPriority := Tc3_DALI.E_DALICommandPriority.Middle );
	IF (NOT fb202QueryDurationTestResult.bBusy) THEN
		fb202QueryDurationTestResult(bStart := FALSE);
		nDurationTestResult := (2 * fb202QueryDurationTestResult.nDurationTestResult);
		nStep := 70;
	END_IF
{endregion}
70:
{region "Query Lamp emergency Time"}
	fb202QueryLampEmergencyTime(	bStart := TRUE,
									nAddress := nAddress,
									eAddressType := Tc3_DALI.E_DALIAddressType.Short,
									eCommandPriority := Tc3_DALI.E_DALICommandPriority.Middle );
	IF (NOT fb202QueryLampEmergencyTime.bBusy) THEN
		fb202QueryLampEmergencyTime(bStart := FALSE);
		nLampEmergencyTime := fb202QueryLampEmergencyTime.nLampEmergencyTime;
		nStep := 75;
	END_IF
{endregion}
75:
{region "Query Lamp total operation Time"}
	fb202QueryLampTotalOperationTime(	bStart := TRUE,
										nAddress := nAddress,
										eAddressType := Tc3_DALI.E_DALIAddressType.Short,
										eCommandPriority := Tc3_DALI.E_DALICommandPriority.Middle );
	IF (NOT fb202QueryLampTotalOperationTime.bBusy) THEN
		fb202QueryLampTotalOperationTime(bStart:= FALSE);
		nLampTotalOperationTime := (4 * fb202QueryLampTotalOperationTime.nLampTotalOperationTime);
		nStep := 80;
	END_IF
{endregion}
80:
{region "Stop Quiescent Mode"}
	fb103StopQuiescentMode(bStart := TRUE,
							eAddressType := Tc3_DALI.E_DALIAddressType.Broadcast,
							eCommandPriority := Tc3_DALI.E_DALICommandPriority.Middle);
	IF (NOT fb103StopQuiescentMode.bBusy) THEN
		fb103StopQuiescentMode(bStart := FALSE);
		nStep := 0;
	END_IF
	{endregion}

{region "Read Status"}
100:
{region "Query Emergency Mode"}
	fb202QueryEmergencyMode(bStart := TRUE,
							nAddress := nAddress,
							eAddressType := Tc3_DALI.E_DALIAddressType.Short,
							eCommandPriority := Tc3_DALI.E_DALICommandPriority.Middle );
	IF (NOT fb202QueryEmergencyMode.bBusy) THEN
		fb202QueryEmergencyMode(bStart:= FALSE);
		sRestMode := SEL(fb202QueryEmergencyMode.nEmergencyMode.0, 'FALSE', 'TRUE');
		sNormalMode := SEL(fb202QueryEmergencyMode.nEmergencyMode.1, 'FALSE', 'TRUE');
		sEmergencyMode := SEL(fb202QueryEmergencyMode.nEmergencyMode.2, 'FALSE', 'TRUE');
		sExtendedEmergency := SEL(fb202QueryEmergencyMode.nEmergencyMode.3, 'FALSE', 'TRUE');
		sFunctionTest := SEL(fb202QueryEmergencyMode.nEmergencyMode.4, 'FALSE', 'TRUE');
		sDurationTest := SEL(fb202QueryEmergencyMode.nEmergencyMode.5, 'FALSE', 'TRUE');
		sHardwiredInhibit := SEL(fb202QueryEmergencyMode.nEmergencyMode.6, 'FALSE', 'TRUE');
		sHardwiredSwitch := SEL(fb202QueryEmergencyMode.nEmergencyMode.7, 'FALSE', 'TRUE');
		nStep := 110;
	END_IF
{endregion}
110:
{region "Query Failure Status"}
	fb202QueryFailureStatus(bStart := TRUE,
							nAddress := nAddress,
							eAddressType := Tc3_DALI.E_DALIAddressType.Short,
							eCommandPriority := Tc3_DALI.E_DALICommandPriority.Middle );
	IF (NOT fb202QueryFailureStatus.bBusy) THEN
		fb202QueryFailureStatus(bStart := FALSE);
		sCircuitFailure := SEL(fb202QueryFailureStatus.nFailureStatus.0, 'FALSE', 'TRUE');
		sBatteryDurationFailure := SEL(fb202QueryFailureStatus.nFailureStatus.1, 'FALSE', 'TRUE');
		sBatteryFailure := SEL(fb202QueryFailureStatus.nFailureStatus.2, 'FALSE', 'TRUE');
		sEmergencyLampFailure := SEL(fb202QueryFailureStatus.nFailureStatus.3, 'FALSE', 'TRUE');
		sFunctionTestExceed := SEL(fb202QueryFailureStatus.nFailureStatus.4, 'FALSE', 'TRUE');
		sDurationTestExceed := SEL(fb202QueryFailureStatus.nFailureStatus.5, 'FALSE', 'TRUE');
		sFunctionTestFailed := SEL(fb202QueryFailureStatus.nFailureStatus.6, 'FALSE', 'TRUE');
		sDurationTestFailed := SEL(fb202QueryFailureStatus.nFailureStatus.7, 'FALSE', 'TRUE');
		nStep := 120;
	END_IF
{endregion}
120:
{region "Query Emergency Status"}
	fb202QueryEmergencyStatus(bStart := TRUE,
							nAddress := nAddress,
							eAddressType := Tc3_DALI.E_DALIAddressType.Short,
							eCommandPriority := Tc3_DALI.E_DALICommandPriority.Middle );
	IF (NOT fb202QueryEmergencyStatus.bBusy) THEN
		fb202QueryEmergencyStatus(bStart := FALSE);
		sInhibitMode := SEL(fb202QueryEmergencyStatus.nEmergencyStatus.0, 'FALSE', 'TRUE');
		sFunctionTestDoneValid := SEL(fb202QueryEmergencyStatus.nEmergencyStatus.1, 'FALSE', 'TRUE');
		sDurationTestDoneValid := SEL(fb202QueryEmergencyStatus.nEmergencyStatus.2, 'FALSE', 'TRUE');
		sBatteryFullCharged := SEL(fb202QueryEmergencyStatus.nEmergencyStatus.3, 'FALSE', 'TRUE');
		sFunctionTestRequestPending := SEL(fb202QueryEmergencyStatus.nEmergencyStatus.4, 'FALSE', 'TRUE');
		sDurationTestRequestPending := SEL(fb202QueryEmergencyStatus.nEmergencyStatus.5, 'FALSE', 'TRUE');
		sIdentificationActive := SEL(fb202QueryEmergencyStatus.nEmergencyStatus.6, 'FALSE', 'TRUE');
		nStep := 0;
	END_IF
{endregion}
{endregion}
{region "Read Parameters"}
200:
	{region "Start Qiescent Mode"}
	fb103StartQuiescentMode(bStart := TRUE,
							eAddressType := Tc3_DALI.E_DALIAddressType.Broadcast,
							eCommandPriority := Tc3_DALI.E_DALICommandPriority.Middle);
	IF (NOT fb103StartQuiescentMode.bBusy) THEN
		fb103StartQuiescentMode(bStart := FALSE);
		nStep := 210;
	END_IF
{endregion}
210:
{region "Query Emergency Level"}
	fb202QueryEmergencyLevel(	bStart := TRUE,
								nAddress := nAddress,
								eAddressType := Tc3_DALI.E_DALIAddressType.Short,
								eCommandPriority := Tc3_DALI.E_DALICommandPriority.Middle );
	IF (NOT fb202QueryEmergencyLevel.bBusy) THEN
		fb202QueryEmergencyLevel (bStart := FALSE);
		nEmergencyLevel := fb202QueryEmergencyLevel.nEmergencyLevel;
		nStep := 220;
	END_IF
{endregion}
220:
{region "Query Emergency Min Level"}
	fb202QueryEmergencyMinLevel(bStart := TRUE,
								nAddress := nAddress,
								eAddressType := Tc3_DALI.E_DALIAddressType.Short,
								eCommandPriority := Tc3_DALI.E_DALICommandPriority.Middle );
	IF (NOT fb202QueryEmergencyMinLevel.bBusy) THEN
		fb202QueryEmergencyMinLevel (bStart := FALSE);
		nEmergencyMinLevel := fb202QueryEmergencyMinLevel.nEmergencyMinLevel;
		nStep := 230;
	END_IF
{endregion}
230:
{region "Query Emergency Max Level"}
	fb202QueryEmergencyMaxLevel(bStart := TRUE,
								nAddress := nAddress,
								eAddressType := Tc3_DALI.E_DALIAddressType.Short,
								eCommandPriority := Tc3_DALI.E_DALICommandPriority.Middle );
	IF (NOT fb202QueryEmergencyMaxLevel.bBusy) THEN
		fb202QueryEmergencyMaxLevel (bStart := FALSE);
		nEmergencyMaxLevel := fb202QueryEmergencyMaxLevel.nEmergencyMaxLevel;
		nStep := 240;
	END_IF
{endregion}
240: 
{region "Query Prolong Time"}
	fb202QueryTestTiming(	bStart := TRUE,
							nAddress := nAddress,
							eAddressType := Tc3_DALI.E_DALIAddressType.Short,
							eCommandPriority := Tc3_DALI.E_DALICommandPriority.Middle,
							eTestTiming:= Tc3_DALI.E_DALITestTiming.ProlongTime);
	IF (NOT fb202QueryTestTiming.bBusy) THEN
		fb202QueryTestTiming (bStart := FALSE);
		nProlongTime := (fb202QueryTestTiming.nValue * 30);
		nStep := 250;
	END_IF
{endregion}
250:
{region "Query Function Test Delay Time"}
	fb202QueryTestTiming(	bStart := TRUE,
							nAddress := nAddress,
							eAddressType := Tc3_DALI.E_DALIAddressType.Short,
							eCommandPriority := Tc3_DALI.E_DALICommandPriority.Middle,
							eTestTiming:= Tc3_DALI.E_DALITestTiming.FunctionTestDelayTime );
	IF (NOT fb202QueryTestTiming.bBusy) THEN
		fb202QueryTestTiming (bStart := FALSE);
		nFunctionTestDelayTime := (fb202QueryTestTiming.nValue * 15);
		fFunctionTestDelayTimeVisu := TO_REAL(nFunctionTestDelayTime)/ 60;
		nStep := 260;
	END_IF
{endregion}
260:
{region "Query Duration Test Delay Time"}
	fb202QueryTestTiming(	bStart := TRUE,
							nAddress := nAddress,
							eAddressType := Tc3_DALI.E_DALIAddressType.Short,
							eCommandPriority := Tc3_DALI.E_DALICommandPriority.Middle,
							eTestTiming := Tc3_DALI.E_DALITestTiming.DurationTestDelayTime);
	IF (NOT fb202QueryTestTiming.bBusy) THEN
		fb202QueryTestTiming (bStart := FALSE);
		nDurationTestDelayTime := (fb202QueryTestTiming.nValue * 15);
		fDurationTestDelayTimeVisu := TO_REAL(nDurationTestDelayTime) / 60;
		nStep := 270;
	END_IF
{endregion}
270:
{region "Query Function Test Interval"}
	fb202QueryTestTiming(	bStart := TRUE,
							nAddress := nAddress,
							eAddressType := Tc3_DALI.E_DALIAddressType.Short,
							eCommandPriority := Tc3_DALI.E_DALICommandPriority.Middle,
							eTestTiming:= Tc3_DALI.E_DALITestTiming.FunctionTestInterval);
	IF (NOT fb202QueryTestTiming.bBusy) THEN
		fb202QueryTestTiming (bStart := FALSE);
		nFunctionTestInterval := fb202QueryTestTiming.nValue;
		nStep := 280;
	END_IF
{endregion}
280:
{region "Query Duration Test Interval"}
	fb202QueryTestTiming(	bStart := TRUE,
							nAddress := nAddress,
							eAddressType := Tc3_DALI.E_DALIAddressType.Short,
							eCommandPriority := Tc3_DALI.E_DALICommandPriority.Middle,
							eTestTiming:= Tc3_DALI.E_DALITestTiming.DurationTestInterval);
	IF (NOT fb202QueryTestTiming.bBusy) THEN
		fb202QueryTestTiming (bStart := FALSE);
		nDurationTestInterval := fb202QueryTestTiming.nValue;
		nStep := 290;
	END_IF
{endregion}
290:
{region "Query Test Execution Timeout"}
	fb202QueryTestTiming(	bStart := TRUE,
							nAddress := nAddress,
							eAddressType := Tc3_DALI.E_DALIAddressType.Short,
							eCommandPriority := Tc3_DALI.E_DALICommandPriority.Middle,
							eTestTiming:= Tc3_DALI.E_DALITestTiming.TestExecutionTimeout);
	IF (NOT fb202QueryTestTiming.bBusy) THEN
		fb202QueryTestTiming (bStart := FALSE);
		nTestExecutionTimeout := fb202QueryTestTiming.nValue;
		nStep := 300;
	END_IF
{endregion}
300:
{region "Query Rated Duration"}
	fb202QueryRatedDuration(bStart := TRUE,
							nAddress := nAddress,
							eAddressType := Tc3_DALI.E_DALIAddressType.Short,
							eCommandPriority := Tc3_DALI.E_DALICommandPriority.Middle );
	IF (NOT fb202QueryRatedDuration.bBusy) THEN
		fb202QueryRatedDuration (bStart := FALSE);
		nRatedDuration := ( 2 * fb202QueryRatedDuration.nRatedDuration);
		nStep := 310;
	END_IF
{endregion}
310:
{region "Query Features"}
	fb202QueryFeatures(	bStart := TRUE,
						nAddress := nAddress,
						eAddressType := Tc3_DALI.E_DALIAddressType.Short,
						eCommandPriority := Tc3_DALI.E_DALICommandPriority.Middle );
	IF (NOT fb202QueryFeatures.bBusy) THEN
		fb202QueryFeatures (bStart := FALSE);
		bIntegralControlGear	:= fb202QueryFeatures.nFeatures.0;
		bMaintainedControlGear	:= fb202QueryFeatures.nFeatures.1;
		bSwitchtedMaintainedControlGear	:= fb202QueryFeatures.nFeatures.2;
		bAutoTestCapability	:= fb202QueryFeatures.nFeatures.3;
		bAdjustableEmergencyLevel	:= fb202QueryFeatures.nFeatures.4;
		bHardwiredInhibitSupported	:= fb202QueryFeatures.nFeatures.5;
		bPhysicalSelectionSupported	:= fb202QueryFeatures.nFeatures.6;
		bRelightinRestModeSupported	:= fb202QueryFeatures.nFeatures.7;
		nStep := 320;
	END_IF
{endregion}
320:
{region "Stop Quiescent Mode"}
	 fb103StopQuiescentMode(bStart := TRUE,
							eAddressType := Tc3_DALI.E_DALIAddressType.Broadcast,
							eCommandPriority := Tc3_DALI.E_DALICommandPriority.Middle);
	IF (NOT fb103StopQuiescentMode.bBusy) THEN
		fb103StopQuiescentMode(bStart := FALSE);
		nStep := 0;
	END_IF
{endregion}
{endregion}
{region "Write Parameters"}
500:
{region "Set Emergency Level"}
	fb202SetEmergencyLevel(	bStart := TRUE,
							nAddress := nAddress,
							eAddressType := Tc3_DALI.E_DALIAddressType.Short,
							eCommandPriority := Tc3_DALI.E_DALICommandPriority.Middle,
							nEmergencyLevel :=  nEmergencyLevel);
	IF (NOT fb202SetEmergencyLevel.bBusy) THEN
		fb202SetEmergencyLevel (bStart := FALSE);
		nStep := 510;
	END_IF
{endregion}
510:
{region "Set Prolong Time"}
	fb202SetProlongTime(	bStart := TRUE,
							nAddress := nAddress,
							eAddressType := Tc3_DALI.E_DALIAddressType.Short,
							eCommandPriority := Tc3_DALI.E_DALICommandPriority.Middle,
							nProlongTime:= TO_BYTE(nProlongTime / 30));
	IF (NOT fb202SetProlongTime.bBusy) THEN
		fb202SetProlongTime (bStart := FALSE);
		nStep := 520;
	END_IF
{endregion}
520:
	nDurationTestDelayTime := TO_UINT((fDurationTestDelayTimeVisu *60) /15);
	fb202SetTestDelayTime(	bStart := TRUE,
							nAddress := nAddress,
							eAddressType := Tc3_DALI.E_DALIAddressType.Short,
							eCommandPriority := Tc3_DALI.E_DALICommandPriority.Middle,
							nTestDelayTime := nDurationTestDelayTime);
	IF (NOT fb202SetTestDelayTime.bBusy) THEN
		fb202SetTestDelayTime (bStart := FALSE);
		nStep := 530;
	END_IF
530:
	fb202SetDurationTestInterval(	bStart := TRUE,
									nAddress := nAddress,
									eAddressType := Tc3_DALI.E_DALIAddressType.Short,
									eCommandPriority := Tc3_DALI.E_DALICommandPriority.Middle,
									nDurationTestInterval := TO_BYTE(nDurationTestInterval));
	IF (NOT fb202SetDurationTestInterval.bBusy) THEN
		fb202SetDurationTestInterval(bStart := FALSE);
		nStep := 540;
	END_IF
{endregion}
{region "Set Function Test Delay time and Function Test Interval"}
540:
	nFunctionTestDelayTime := TO_UINT(fFunctionTestDelayTimeVisu * 60 / 15);
	fb202SetTestDelayTime(	bStart := TRUE,
							nAddress := nAddress,
							eAddressType := Tc3_DALI.E_DALIAddressType.Short,
							eCommandPriority := Tc3_DALI.E_DALICommandPriority.Middle,
							nTestDelayTime := nFunctionTestDelayTime);
	IF (NOT fb202SetTestDelayTime.bBusy) THEN
		fb202SetTestDelayTime(bStart := FALSE);
		nStep := 550;
	END_IF
550:
	fb202SetFunctionTestInterval(	bStart := TRUE,
									nAddress := nAddress,
									eAddressType := Tc3_DALI.E_DALIAddressType.Short,
									eCommandPriority := Tc3_DALI.E_DALICommandPriority.Middle,
									nFunctionTestInterval := TO_BYTE(nFunctionTestInterval));
	IF (NOT fb202SetFunctionTestInterval.bBusy) THEN
		fb202SetFunctionTestInterval (bStart := FALSE);
		nStep := 560;
	END_IF
{endregion}
560:
{region "Set Test Execution Timeout"}
	fb202SetTestExecutionTimeout(	bStart := TRUE,
									nAddress := nAddress,
									eAddressType := Tc3_DALI.E_DALIAddressType.Short,
									eCommandPriority := Tc3_DALI.E_DALICommandPriority.Middle,
									nTestExecutionTimeout := TO_BYTE(nTestExecutionTimeout));
	IF (NOT fb202SetTestExecutionTimeout.bBusy) THEN
		fb202SetTestExecutionTimeout (bStart := FALSE);
		nStep := 0;
	END_IF
{endregion}
{endregion}
END_CASE

END_FUNCTION_BLOCK

// ---- POUs/DALI/DALI_Setup/FBs/FB_Part208Switching.TcPOU
FUNCTION_BLOCK FB_Part208Switching
VAR_INPUT
	ipDALICommunication					:	I_DALICommunication;
END_VAR
VAR_OUTPUT
	bBusy								:	BOOL;
END_VAR
VAR
	{region "Visu"}
	bRead								:	BOOL;
	bWrite								:	BOOL;
	sGearType							:	STRING[80];
	bThreshold							:	BOOL;
	bAddressingPhysical					:	BOOL;
	nDownSwitchOffThreshold				:	BYTE;
	nDownSwitchOnThreshold				:	BYTE;
	nUpSwitchOffThreshold				:	BYTE;
	nUpSwitchOnThreshold				:	byte;
	{endregion}
	nStep								:	INT;
	nAddress							:	BYTE;
	bHideWaitSymbol						:	BOOL := TRUE;
	nGearType							:	BYTE;

	fb103StartQuiescentMode				:	FB_DALI103StartQuiescentMode(0);
	fb103StopQuiescentMode				:	FB_DALI103StopQuiescentMode(0);
	fb208QueryGearType					:	FB_DALI208QueryGearType(0);
	fb208QueryFeatures					:	FB_DALI208QueryFeatures(0);
	fb208QuerySwitchStatus				:	FB_DALI208QuerySwitchStatus(0);
	fb208QueryDownSwitchOffThreshold	:	FB_DALI208QueryDownSwitchOffThreshold(0);
	fb208QueryDownSwitchOnThreshold		:	FB_DALI208QueryDownSwitchOnThreshold(0);
	fb208QueryUpSwitchOffThreshold		:	FB_DALI208QueryUpSwitchOffThreshold(0);
	fb208QueryUpSwitchOnThreshold		:	FB_DALI208QueryUpSwitchOnThreshold(0);
	fb208SetDownSwitchOffThreshold		:	FB_DALI208SetDownSwitchOffThreshold(0);
	fb208SetDownSwitchOnThreshold		:	FB_DALI208SetDownSwitchOnThreshold(0);
	fb208SetUpSwitchOffThreshold		:	FB_DALI208SetUpSwitchOffThreshold(0);
	fb208SetUpSwitchOnThreshold			:	FB_DALI208SetUpSwitchOnThreshold(0);
END_VAR

{region "Detect Commands"}
IF (bRead AND (nStep = 0)) THEN
	nStep := 5;
	bRead := FALSE;
	bHideWaitSymbol := FALSE;
END_IF

IF (bWrite AND (nStep = 0)) THEN
	nStep := 500;
	bWrite := FALSE;
	bHideWaitSymbol := FALSE;
END_IF
{endregion}
{region "Manage Dialog Selection}
IF (nStep = 0) THEN
	bBusy := FALSE;
ELSE
	bBusy := TRUE;
END_IF
{endregion}
{region "Execute Commands"}
CASE nStep OF
0:
{region "Init"}
	bRead := FALSE;
	bWrite := FALSE;
	bHideWaitSymbol := TRUE;

	fb103StartQuiescentMode.ipDALICommunication := ipDALICommunication;
	fb103StopQuiescentMode.ipDALICommunication := ipDALICommunication;
	fb208QueryGearType.ipDALICommunication := ipDALICommunication;
	fb208QueryFeatures.ipDALICommunication := ipDALICommunication;
	fb208QuerySwitchStatus.ipDALICommunication := ipDALICommunication;
	fb208QueryDownSwitchOffThreshold.ipDALICommunication := ipDALICommunication;
	fb208QueryDownSwitchOnThreshold.ipDALICommunication := ipDALICommunication;
	fb208QueryUpSwitchOffThreshold.ipDALICommunication := ipDALICommunication;
	fb208QueryUpSwitchOnThreshold.ipDALICommunication := ipDALICommunication;
	fb208SetDownSwitchOffThreshold.ipDALICommunication := ipDALICommunication;
	fb208SetDownSwitchOnThreshold.ipDALICommunication := ipDALICommunication;
	fb208SetUpSwitchOffThreshold.ipDALICommunication := ipDALICommunication;
	fb208SetUpSwitchOnThreshold.ipDALICommunication := ipDALICommunication;
{endregion}
{region "Read"}
5:
{region "Start Qiescent Mode"}
	fb103StartQuiescentMode(bStart := TRUE,
							eAddressType := Tc3_DALI.E_DALIAddressType.Broadcast,
							eCommandPriority := Tc3_DALI.E_DALICommandPriority.Middle);
	IF (NOT fb103StartQuiescentMode.bBusy) THEN
		fb103StartQuiescentMode(bStart := FALSE);
		nStep := 10;
	END_IF
{endregion}
10:
{region "Query Gear Type"}
	fb208QueryGearType(	bStart := TRUE,
						nAddress := nAddress,
						eAddressType := Tc3_DALI.E_DALIAddressType.Short,
						eCommandPriority := Tc3_DALI.E_DALICommandPriority.Middle,
						nGearType => nGearType);
	IF (NOT fb208QueryGearType.bBusy) THEN
		fb208QueryGearType(bStart := FALSE);
		sGearType := GearType(nGearType := nGearType);
		nStep := 20;
	END_IF
{endregion}
20:
{region "Query Features"}
	fb208QueryFeatures(	bStart := TRUE,
						nAddress := nAddress,
						eAddressType := Tc3_DALI.E_DALIAddressType.Short,
						eCommandPriority := Tc3_DALI.E_DALICommandPriority.Middle);
	IF (NOT fb208QueryFeatures.bBusy) THEN
		fb208QueryFeatures(bStart := FALSE);
		bThreshold := fb208QueryFeatures.nFeatures.3;
		bAddressingPhysical := fb208QueryFeatures.nFeatures.7;
		nStep := 30;
	END_IF
{endregion}
30:
{region "Query Down Switch Off Threshold"}
	fb208QueryDownSwitchOffThreshold(	bStart := TRUE,
										nAddress := nAddress,
										eAddressType := Tc3_DALI.E_DALIAddressType.Short,
										eCommandPriority := Tc3_DALI.E_DALICommandPriority.Middle);
	IF (NOT fb208QueryDownSwitchOffThreshold.bBusy) THEN
		fb208QueryDownSwitchOffThreshold(bStart := FALSE);
		nDownSwitchOffThreshold := fb208QueryDownSwitchOffThreshold.nDownSwitchOffThreshold;
		nStep := 40;
	END_IF
{endregion}
40:
{region "Query Down Switch On Threshold"}
	fb208QueryDownSwitchOnThreshold(bStart := TRUE,
									nAddress := nAddress,
									eAddressType := Tc3_DALI.E_DALIAddressType.Short,
									eCommandPriority := Tc3_DALI.E_DALICommandPriority.Middle);
	IF (NOT fb208QueryDownSwitchOnThreshold.bBusy) THEN
		fb208QueryDownSwitchOnThreshold(bStart := FALSE);
		nDownSwitchOnThreshold := fb208QueryDownSwitchOnThreshold.nDownSwitchOnThreshold;
		nStep := 50;
	END_IF
{endregion}
50:
{region "Query Up Switch Off Threshold"}
	fb208QueryUpSwitchOffThreshold(	bStart := TRUE,
									nAddress := nAddress,
									eAddressType := Tc3_DALI.E_DALIAddressType.Short,
									eCommandPriority := Tc3_DALI.E_DALICommandPriority.Middle);
	IF (NOT fb208QueryUpSwitchOffThreshold.bBusy) THEN
		fb208QueryUpSwitchOffThreshold(bStart := FALSE);
		nUpSwitchOffThreshold := fb208QueryUpSwitchOffThreshold.nUpSwitchOffThreshold;
		nStep := 60;
	END_IF
{endregion}
60:
{region "Query Up Switch On Threshold"}
	fb208QueryUpSwitchOnThreshold(	bStart := TRUE,
									nAddress := nAddress,
									eAddressType := Tc3_DALI.E_DALIAddressType.Short,
									eCommandPriority := Tc3_DALI.E_DALICommandPriority.Middle );
	IF (NOT fb208QueryUpSwitchOnThreshold.bBusy) THEN
		fb208QueryUpSwitchOnThreshold(bStart := FALSE);
		nUpSwitchOnThreshold := fb208QueryUpSwitchOnThreshold.nUpSwitchOnThreshold;
		nStep := 70;
	END_IF
{endregion}
70:
{region "Stop Qiescent Mode"}
	fb103StopQuiescentMode(	bStart := TRUE,
							eAddressType := Tc3_DALI.E_DALIAddressType.Broadcast,
							eCommandPriority := Tc3_DALI.E_DALICommandPriority.Middle);
	IF (NOT fb103StopQuiescentMode.bBusy) THEN
		fb103StopQuiescentMode(bStart:= FALSE);
		nStep := 0;
	END_IF
{endregion}
{region "Write"}
500:
{region "Set Down Switch Off Threshold"}
	fb208SetDownSwitchOffThreshold(	bStart := TRUE,
									nAddress := nAddress,
									eAddressType := Tc3_DALI.E_DALIAddressType.Short,
									eCommandPriority := Tc3_DALI.E_DALICommandPriority.Middle,
									nDownSwitchOffThreshold := nDownSwitchOffThreshold);
	IF (NOT fb208SetDownSwitchOffThreshold.bBusy) THEN
		fb208SetDownSwitchOffThreshold(bStart := FALSE);
		nStep := 510;
	END_IF
{endregion}
510:
{region "Set Down Switch On Threshold"}
	fb208SetDownSwitchOnThreshold(	bStart := TRUE,
									nAddress := nAddress,
									eAddressType := Tc3_DALI.E_DALIAddressType.Short,
									eCommandPriority := Tc3_DALI.E_DALICommandPriority.Middle,
									nDownSwitchOnThreshold := nDownSwitchOnThreshold);
	IF (NOT fb208SetDownSwitchOnThreshold.bBusy) THEN
		fb208SetDownSwitchOnThreshold(bStart := FALSE);
		nStep := 520;
	END_IF
{endregion}
520:
{region "Set Up Switch Off Threshold"}
	fb208SetUpSwitchOffThreshold(	bStart := TRUE,
									nAddress := nAddress,
									eAddressType := Tc3_DALI.E_DALIAddressType.Short,
									eCommandPriority := Tc3_DALI.E_DALICommandPriority.Middle,
									nUpSwitchOffThreshold := nUpSwitchOffThreshold);
	IF (NOT fb208SetUpSwitchOffThreshold.bBusy) THEN
		fb208SetUpSwitchOffThreshold(bStart := FALSE);
		nStep := 530;
	END_IF
{endregion}
530:
{region "Set Up Switch On Threshold"}
	fb208SetUpSwitchOnThreshold(bStart := TRUE,
								nAddress := nAddress,
								eAddressType := Tc3_DALI.E_DALIAddressType.Short,
								eCommandPriority := Tc3_DALI.E_DALICommandPriority.Middle,
								nUpSwitchOnThreshold := nUpSwitchOnThreshold);
	IF (NOT fb208SetUpSwitchOnThreshold.bBusy) THEN
		fb208SetUpSwitchOnThreshold(bStart := FALSE);
		nStep := 0;
	END_IF
{endregion}
{endregion}
END_CASE
{endregion}

END_FUNCTION_BLOCK

// ---- POUs/DALI/DALI_Setup/FBs/FB_Part301PushButton.TcPOU
FUNCTION_BLOCK FB_Part301PushButton
VAR_INPUT
	ipDALICommunication			:	I_DALICommunication;
END_VAR
VAR_OUTPUT
	bBusy						:	BOOL;
END_VAR
VAR
	{region "Visu"}
	sInputValue					:	STRING[25];
	nInstanceError				:	BYTE;
	nResolution					:	BYTE;
	eEventScheme				:	E_DALIEventScheme;
	nEventFilter				:	DWORD;
	nRepeat						:	UINT(100..2000);
	nStuck						:	BYTE(5..255);
	nShort						:	UINT(0..5100);
	nShortMin					:	UINT;
	nDouble						:	UINT(0..2000);
	nDoubleMin					:	UINT;
	bRead						:	BOOL;
	bWrite						:	BOOL;
	bEnable						:	BOOL;
	bButtonReleased				:	BOOL;
	bButtonPressed				:	BOOL;
	bShortPress					:	BOOL;
	bDoublePress				:	BOOL;
	bLongPressStart				:	BOOL;
	bLongPressRepeat			:	BOOL;
	bLongPressStop				:	BOOL;
	bButtonStuck				:	BOOL;
	bNoRepeatTimer				:	BOOL;
	bNoStuckTimer				:	BOOL;
	bNoShortTimer				:	BOOL;
	bNoDoubleTimer				:	BOOL;
	eEventPriority				:	E_DALIEventPriority := E_DALIEventPriority.Middle;
{endregion}
	nStep						:	INT;
	nAddress					:	BYTE;
	nInstanceAddress			:	BYTE;
	bHideWaitSymbol				:	BOOL := TRUE;
	nInputValue					:	LWORD;
	nAddressInfo01				:	BYTE;
	nAddressInfo02				:	BYTE;

	fbGetInputNotification		:	FB_DALIGetInputNotification(0);
	fb103StartQuiescentMode		:	FB_DALI103StartQuiescentMode(0);
	fb103StopQuiescentMode		:	FB_DALI103StopQuiescentMode(0);
	fb103QueryInstanceError		:	FB_DALI103QueryInstanceError(0);
	fb103QueryInstanceStatus	:	FB_DALI103QueryInstanceStatus(0);
	fb103QueryResolution		:	FB_DALI103QueryResolution(0);
	fb103QueryInputValue		:	FB_DALI103QueryInputValue(0);
	fb103QueryEventScheme		:	FB_DALI103QueryEventScheme(0);
	fb103QueryEventFilter		:	FB_DALI103QueryEventFilter(0);
	fb103QueryEventPriority		:	FB_DALI103QueryEventPriority(0);
	fb301QueryRepeatTimer		:	FB_DALI301QueryRepeatTimer(0);
	fb301QueryStuckTimer		:	FB_DALI301QueryStuckTimer(0);
	fb301QueryShortTimer		:	FB_DALI301QueryShortTimer(0);
	fb301QueryShortTimerMin		:	FB_DALI301QueryShortTimerMin(0);
	fb301QueryDoubleTimer		:	FB_DALI301QueryDoubleTimer(0);
	fb301QueryDoubleTimerMin	:	FB_DALI301QueryDoubleTimerMin(0);
	fb103EnableInstance			:	FB_DALI103EnableInstance(0);
	fb103DisableInstance		:	FB_DALI103DisableInstance(0);
	fb103SetEventScheme			:	FB_DALI103SetEventScheme(0);
	fb103SetEventFilter			:	FB_DALI103SetEventFilter(0);
	fb103SetEventPriority		:	FB_DALI103SetEventPriority(0);
	fb301SetRepeatTimer			:	FB_DALI301SetRepeatTimer(0);
	fb301SetStuckTimer			:	FB_DALI301SetStuckTimer(0);
	fb301SetShortTimer			:	FB_DALI301SetShortTimer(0);
	fb301SetDoubleTimer			:	FB_DALI301SetDoubleTimer(0);
END_VAR

{region "Detect Commands"}
IF (bRead AND (nStep = 0)) THEN
	nStep := 5;
	bRead := FALSE;
	bHideWaitSymbol := FALSE;
END_IF

IF (bWrite AND (nStep = 0)) THEN
	nStep := 1000;
	bWrite := FALSE;
	bHideWaitSymbol := FALSE;
END_IF
{endregion}
{region "Manage Dialog Selection}
IF (nStep = 0) THEN
	bBusy := FALSE;
ELSE
	bBusy := TRUE;
END_IF
{endregion}
{region "Execute Commands"}
CASE nStep OF
0:
{region "Init"}
	bRead := FALSE;
	bWrite := FALSE;
	bHideWaitSymbol := TRUE;

	fbGetInputNotification.ipDALICommunication := ipDALICommunication;
	fb103StartQuiescentMode.ipDALICommunication := ipDALICommunication;
	fb103StopQuiescentMode.ipDALICommunication := ipDALICommunication;
	fb103QueryInstanceError.ipDALICommunication := ipDALICommunication;
	fb103QueryInstanceStatus.ipDALICommunication := ipDALICommunication;
	fb103QueryResolution.ipDALICommunication := ipDALICommunication;
	fb103QueryInputValue.ipDALICommunication := ipDALICommunication;
	fb103QueryEventScheme.ipDALICommunication := ipDALICommunication;
	fb103QueryEventFilter.ipDALICommunication := ipDALICommunication;
	fb103QueryEventPriority.ipDALICommunication := ipDALICommunication;
	fb301QueryRepeatTimer.ipDALICommunication := ipDALICommunication;
	fb301QueryStuckTimer.ipDALICommunication := ipDALICommunication;
	fb301QueryShortTimer.ipDALICommunication := ipDALICommunication;
	fb301QueryShortTimerMin.ipDALICommunication := ipDALICommunication;
	fb301QueryDoubleTimer.ipDALICommunication := ipDALICommunication;
	fb301QueryDoubleTimerMin.ipDALICommunication := ipDALICommunication;
	fb103EnableInstance.ipDALICommunication := ipDALICommunication;
	fb103DisableInstance.ipDALICommunication := ipDALICommunication;
	fb103SetEventScheme.ipDALICommunication := ipDALICommunication;
	fb103SetEventFilter.ipDALICommunication := ipDALICommunication;
	fb103SetEventPriority.ipDALICommunication := ipDALICommunication;
	fb301SetRepeatTimer.ipDALICommunication := ipDALICommunication;
	fb301SetStuckTimer.ipDALICommunication := ipDALICommunication;
	fb301SetShortTimer.ipDALICommunication := ipDALICommunication;
	fb301SetDoubleTimer.ipDALICommunication := ipDALICommunication;
{endregion}
{region "Read Notifications"}
	CASE eEventScheme OF
	0:
		nAddressInfo01 := 1;
		nAddressInfo02 := nInstanceAddress;
	1:
		nAddressInfo01 := nAddress;
		nAddressInfo02 := 1;
	2:
		nAddressInfo01 := nAddress;
		nAddressInfo02 := nInstanceAddress;
	END_CASE

